					BACnetCalendarEntryType_DateRange:
						(* caclulate event entry size and write into data structure *)
						_pSpEventCalEntryRange^.nEntrySize :=	_cbTotalEntry
															+	SIZEOF(_pSpEventCalEntryRange^.stListEntry.eEventChoice)
															+	SIZEOF(_pSpEventCalEntryRange^.stListEntry.iEventPriority)
															+	SIZEOF(_pSpEventCalEntryRange^.stListEntry.nRes1)
															+	SIZEOF(_pSpEventCalEntryRange^.stListEntry.nRes2)
															+	SIZEOF(_pSpEventCalEntryRange^.stListEntry.stCalEntry);
						(* copy event data *)
						_pSpEventCalEntryRange^.stListEntry.eEventChoice := BACnetSpecialEventChoice_calendarEntry;
						_pSpEventCalEntryRange^.stListEntry.nRes1 := 0;
						_pSpEventCalEntryRange^.stListEntry.iEventPriority := stExceptSched.arrEntries[_iEntry].ePriority;
						_pSpEventCalEntryRange^.stListEntry.stCalEntry.eEntryChoice := BACnetCalendarEntryChoice_dateRange;
						_pSpEventCalEntryRange^.stListEntry.stCalEntry.nRes := 0;
						_pSpEventCalEntryRange^.stListEntry.stCalEntry.stStartDate := stExceptSched.arrEntries[_iEntry].stDate.stStart;
						_pSpEventCalEntryRange^.stListEntry.stCalEntry.stEndDate := stExceptSched.arrEntries[_iEntry].stDate.stEnd;

					BACnetCalendarEntryType_WeekNDay:
						(* caclulate event entry size and write into data structure *)
						_pSpEventCalEntryWnD^.nEntrySize :=	_cbTotalEntry
															+	SIZEOF(_pSpEventCalEntryWnD^.stListEntry.eEventChoice)
															+	SIZEOF(_pSpEventCalEntryWnD^.stListEntry.iEventPriority)
															+	SIZEOF(_pSpEventCalEntryWnD^.stListEntry.nRes1)
															+	SIZEOF(_pSpEventCalEntryWnD^.stListEntry.nRes2)
															+	SIZEOF(_pSpEventCalEntryWnD^.stListEntry.nRes3)
															+	SIZEOF(_pSpEventCalEntryWnD^.stListEntry.stCalEntry);
						(* copy event data *)
						_pSpEventCalEntryWnD^.stListEntry.eEventChoice := BACnetSpecialEventChoice_calendarEntry;
						_pSpEventCalEntryWnD^.stListEntry.nRes1 := 0;
						_pSpEventCalEntryWnD^.stListEntry.iEventPriority := stExceptSched.arrEntries[_iEntry].ePriority;
						_pSpEventCalEntryWnD^.stListEntry.stCalEntry.eEntryChoice := BACnetCalendarEntryChoice_weekNDay;
						_pSpEventCalEntryWnD^.stListEntry.stCalEntry.nRes1 := 0;
						_pSpEventCalEntryWnD^.stListEntry.stCalEntry.iDay := stExceptSched.arrEntries[_iEntry].stWeekNDay.iDay;
						_pSpEventCalEntryWnD^.stListEntry.stCalEntry.iMonth := stExceptSched.arrEntries[_iEntry].stWeekNDay.iMonth;
						_pSpEventCalEntryWnD^.stListEntry.stCalEntry.iWeekOfMonth := stExceptSched.arrEntries[_iEntry].stWeekNDay.iWeekOfMonth;

					BACnetCalendarEntryType_Ref:
						(* caclulate event entry size and write into data structure *)
						_pSpEventCalRef^.nEntrySize :=	_cbTotalEntry
													+	SIZEOF(_pSpEventCalRef^.stListEntry.eEventChoice)
													+	SIZEOF(_pSpEventCalRef^.stListEntry.iEventPriority)
													+	SIZEOF(_pSpEventCalRef^.stListEntry.nRes1)
													+	SIZEOF(_pSpEventCalRef^.stListEntry.nRes2)
													+	SIZEOF(_pSpEventCalRef^.stListEntry.nRes3)
													+	SIZEOF(_pSpEventCalRef^.stListEntry.nRes4)
													+	SIZEOF(_pSpEventCalRef^.stListEntry.tCalRef);
						(* copy event data *)
						_pSpEventCalRef^.stListEntry.eEventChoice := BACnetSpecialEventChoice_calendarReference;
						_pSpEventCalRef^.stListEntry.nRes1 := 0;
						_pSpEventCalRef^.stListEntry.iEventPriority := stExceptSched.arrEntries[_iEntry].ePriority;
						_pSpEventCalRef^.stListEntry.tCalRef := stExceptSched.arrEntries[_iEntry].stCalRef.tCalObjectId;

				END_CASE

				(* set next entry flag *)
				IF (_pOldEventEntrySize <> 0) THEN
					_pOldEventEntrySize^ := _pOldEventEntrySize^ + 16#80000000;
				END_IF

				(* next calendar entry *)
				_NextEvent();
			END_IF

		END_FOR

		(* send data *)
		_i := 19;

	19:
		IF _fbWriteProp.bExecute AND (NOT _fbWriteProp.bBusy) THEN
			(* check result *)
			_fbWriteProp.bExecute := FALSE;
			IF _fbWriteProp.bError THEN
				nErrorId := BACnet_ERR_ADS_Write;
			ELSE
				stExceptSched.nSet := stExceptSched.nSet +1;
			END_IF
			_i := 100;
		ELSE
			(* start ADS write *)
			_fbWriteProp.bExecute := TRUE;
		END_IF

	100: (* Done *)
		bDone := (nErrorId = BACnet_ERR_NO_ERROR);
		(* release ADS buffer *)
		stBACnet_AdsBuffer.iLocked := 0;
		(* release data array *)
		stExceptSched.bBusy := FALSE;
		(* go idle *)
		_i := 0;

END_CASE

(* set error flag *)
bError 	:= nErrorId > BACnet_ERR_NO_ERROR;
bBusy 	:= _i > 0;
END_FUNCTION_BLOCK
ACTION _NextEvent:
_bNextEvent := ((_pSpEventCalEntryDate^.nEntrySize AND 16#80000000) = 16#80000000);
_cbTmpSize := _F_BACnet_AlignedSize(_pSpEventCalEntryDate^.nEntrySize AND 16#7FFFFFFF) + SIZEOF(_pSpEventCalEntryDate^.nEntrySize) + SIZEOF(_pSpEventCalEntryDate^.nRes);
_pOldEventEntrySize		:= ADR(_pSpEventCalEntryDate^.nEntrySize);
_pSpEventCalEntryDate	:= _pSpEventCalEntryDate + _cbTmpSize;
_pSpEventCalEntryRange	:= _pSpEventCalEntryRange + _cbTmpSize;
_pSpEventCalEntryWnD	:= _pSpEventCalEntryWnD + _cbTmpSize;
_pSpEventCalRef			:= _pSpEventCalRef + _cbTmpSize;
_cbTotalBuf := _cbTotalBuf + _cbTmpSize;
_pOldTimeValue := 0;
END_ACTION
ACTION _NextTimeValue:
_bNextTimeValue := (_pTimeValue^.nEntrySize AND 16#80000000) = 16#80000000;
_cbTmpSize := 	(_F_BACnet_AlignedSize(_pTimeValue^.nEntrySize) AND 16#7FFFFFFF)
			+	SIZEOF(_pTimeValue^.nEntrySize)
			+	SIZEOF(_pTimeValue^.nRes);
_pOldTimeValue := _pTimeValue;
_pTimeValue := _pTimeValue + _cbTmpSize;
END_ACTION

(* POU FB_BACnet_ExceptionSchedulePropertyReal, ST *)
FUNCTION_BLOCK FB_BACnet_ExceptionSchedulePropertyReal
VAR_INPUT
	tObjectID			: T_BACnet_ObjectIdentifier := 16#FFFFFFFF;
	bAutoGet			: BOOL:=TRUE; (* TRUE = get data from property when ADS connection OR object ID changed *)
	bGet				: BOOL; (* FALSE --> TRUE = get data from property *)
	bSet				: BOOL; (* FALSE --> TRUE = set data into property *)
END_VAR
VAR_IN_OUT
	stExceptSched		: ST_BACnet_ExceptionScheduleReal;
	stAdsConn			: ST_BACnet_AdsConnection;
END_VAR
VAR_OUTPUT
	bDone				: BOOL;
	bBusy				: BOOL;
	bError				: BOOL;
	nErrorId			: UINT;
END_VAR
VAR
	_fbReadProp		: FB_BACnet_ReadProp;
	_fbWriteProp	: FB_BACnet_WriteProp;
	_i				: INT;
	_rtrigGet		: R_TRIG;
	_rtrigSet		: R_TRIG;

	_pOldEventEntrySize		: POINTER TO DWORD;
	_pSpEventCalEntryDate	: POINTER TO ST_BACnet_SpecialEventListCalEntryDate;
	_pSpEventCalEntryRange	: POINTER TO ST_BACnet_SpecialEventListCalEntryRange;
	_pSpEventCalEntryWnD	: POINTER TO ST_BACnet_SpecialEventListCalEntryWnD;
	_pSpEventCalRef			: POINTER TO ST_BACnet_SpecialEventListCalReference;
	_pTimeValue		: POINTER TO ST_BACnet_TimeValueList;
	_pOldTimeValue	: POINTER TO ST_BACnet_TimeValueList;

	_iEntry			: INT;
	_iTv			: INT;

	_bNextEvent		: BOOL;
	_bNextTimeValue	: BOOL;

	_cbTmpSize		: UDINT;
	_cbTotalEntry	: UDINT;
	_cbTotalBuf		: UDINT;
	_nAdsReloadOld	: USINT;
	_tObjectIDOld	: T_BACnet_ObjectIdentifier := 16#FFFFFFFF;

	_pReal			: POINTER TO REAL;
END_VAR
(*

Listheader:

typedef struct _ListEntryHdr
{
      DWORD nEntrySize;
      DWORD hdrInfo;
}ListEntryHdr, *PListEntryHdr;

#define ListAlignedSize(n)         (4*(((n)+3)/4))
#define FirstListEntry(p) ( (p)->nEntrySize == 0 )                          ? NULL:p
#define NextListEntry(p) ( ( ((p)->nEntrySize&0x80000000) == 0 ) ? NULL:(PBYTE)(p) + ( ListAlignedSize((p)->nEntrySize&~(0x80000000)) + sizeof(ListEntryHdr)) ) // +4 da für nEntrySize 4 Byte reserviert sind, HighBit ausmaskieren
#define ElemSize(p) ((p)->nEntrySize&(~0x80000000))
#define AlignedEntrySize(p) (ListAlignedSize((p)->nEntrySize&(~0x80000000)))

###################################################################

PropExceptionSchedule:

enum BACnetSpecialEventChoice
{
      calendarEntry,
      calendarReference,
      MaxBACnetSpecialEventChoice
};

typedef struct _BACnetCalendarEntry
{
      BACnetCalendarEntryChoice choice;
      union
      {
            BACnetDate              date;
            BACnetDateRange   dateRange;
            BACnetWeekNDay          weekNDay;
      };
}BACnetCalendarEntry, *PBACnetCalendarEntry;

enum BACnetValueChoice
{
      NullValue                    = 0,
      BoolValue                    = 1,
      UnsignedValue                = 2,
      SignedValue                  = 3,
      RealValue                    = 4,
      DoubleValue                  = 5,
      OctedStringValue        = 6,
      CharStringValue         = 7,
      ObjectIdentifierValue = 8,   // but DataType is 0x0C
      EnumerationValue        = 9,
      MaxBACnetValueChoice    = 10
};

typedef struct _BACnetValue  
{
      BACnetValueChoice choice;
      DWORD                        length;     // Alignment + Datenlänge die folgt
      union
      {
            BOOL                                     boolValue;
            FLOAT                                    realValue;
            DOUBLE                                   doubleValue;
            INT                                      signedValue;
            UINT                                     unsignedValue;
            BYTE*                                    pOctedStringValue; 
            CHAR*                                    pCharStringValue;
            BACnetObjectIdentifier  objectIdentifierValue;
            EnumerationValueType         enumerationValue;
      };
}BACnetValue, *PBACnetValue;

typedef struct _BACnetTimeValue
{
      BACnetTime time;
      DWORD  reserved;  // 64bit Alignment
      BACnetValue value;
}BACnetTimeValue, *PBACnetTimeValue;

typedef struct _BACnetTimeValueList
{
      DWORD nEntrySize; // 0x80000000 -> next entry
      DWORD reserved;
      BACnetTimeValue listEntry;
}BACnetTimeValueList, *PBACnetTimeValueList;

typedef struct _BACnetSpecialEvent
{
      BACnetSpecialEventChoice choice;
      union
      {
            BACnetCalendarEntry calendarEntry;
            BACnetObjectIdentifier calendarReference;
      };
      DWORD eventPriority; // DWORD due to alignment
      DWORD reserved;
      BACnetTimeValueList listOfTimeValues;
}BACnetSpecialEvent, *PBACnetSpecialEvent;

typedef struct _BACnetSpecialEventList
{
      DWORD nEntrySize; // 0x80000000 -> next entry
      DWORD reserved;
      BACnetSpecialEvent listEntry;
}BACnetSpecialEventList, *PBACnetSpecialEventList;

###################################################################

PropWeeklySchedule:

typedef struct _BACnetDailySchedule
{
      DWORD nEntrySize; // 0x80000000 -> next entry
      DWORD reserved;
      BACnetTimeValueList listEntry;
} BACnetDailySchedule, *PBACnetDailySchedule;

###################################################################

PropScheduleDefault / PropPresentValue

typedef struct _BACnetValueList
{
      DWORD nEntrySize; // 0x80000000 -> next entry
      DWORD reserved;
      BACnetValue listEntry;
} BACnetValueList, *PBACnetValueList;

###################################################################

*)

(* ADS read *)
_fbReadProp(
	BACnetDevicePort	:= stAdsConn.nAmsPort,
	bExecute			:= ,
	sNetId				:= stAdsConn.sAmsNetId,
	ObjectType			:= F_BACnet_GetObjType(tObjectID),
	PropertyID			:= BACnetPropertyIdentifier_ExceptionSchedule,
	DataType			:= BACnetDataType_SpecialEventList,
	ObjectInstance		:= F_BACnet_GetObjInstance(tObjectID),
	ptrValue			:= ADR(stBACnet_AdsBuffer.arrData),
	nLenValue			:= SIZEOF(stBACnet_AdsBuffer.arrData),
	bDone				=> ,
	bBusy				=> ,
	bError				=> ,
	nErrID				=> ,
	nProcessedLen		=> );

(* ADS write *)
_fbWriteProp(
	BACnetDevicePort	:= stAdsConn.nAmsPort,
	bExecute			:= ,
	sNetId				:= stAdsConn.sAmsNetId,
	ObjectType			:= F_BACnet_GetObjType(tObjectID),
	PropertyID			:= BACnetPropertyIdentifier_ExceptionSchedule,
	Priority			:= BACnetPriority_None,
	DataType			:= BACnetDataType_SpecialEventList,
	ObjectInstance		:= F_BACnet_GetObjInstance(tObjectID),
	ptrValue			:= ADR(stBACnet_AdsBuffer.arrData),
	nLenValue			:= _cbTotalBuf,
	bDone				=> ,
	bBusy				=> ,
	bError				=> ,
	nErrID				=> );

(* trigger start event *)
_rtrigGet(CLK:= bGet, Q=> );
_rtrigSet(CLK:= bSet, Q=> );

(* state machine *)
CASE _i OF

	0: (* Idle *)
		IF 		_rtrigGet.Q
			OR	_rtrigSet.Q
			OR	(		(		(_nAdsReloadOld <> stAdsConn.nReload)
							OR	(_tObjectIDOld <> tObjectID)
						)
					AND	bAutoGet
				)
			OR	stExceptSched.bReqGet
			OR	stExceptSched.bReqSet
		THEN
			IF (NOT stAdsConn.bValid) THEN
				(* ADS connection not valid *)
				nErrorId := BACnet_ERR_INVALID_ADS_CONN;
			ELSIF (NOT stAdsConn.bServer AND NOT stAdsConn.bClient) THEN
				(* not a server nor a client *)
				nErrorId := BACnet_ERR_ADS_NoServerClient;
			ELSE
				(* decide get or set *)
				IF _rtrigGet.Q OR stExceptSched.bReqGet  THEN
					_i := 1;
					stExceptSched.bReqGet := FALSE;
				ELSIF _rtrigSet.Q OR stExceptSched.bReqSet THEN
					_i := 11;
					stExceptSched.bReqSet := FALSE;
				ELSIF bAutoGet THEN
					_i := 1;
					stExceptSched.bReqGet := FALSE;
				END_IF
				nErrorId := BACnet_ERR_NO_ERROR;
				(* reset index *)
				_iEntry		:= 0;
				(* remind parameter *)
				_tObjectIDOld := tObjectID;
				_nAdsReloadOld := stAdsConn.nReload;
				(* lock data array *)
				stExceptSched.bBusy := TRUE;
			END_IF
			(* reset done flag *)
			bDone := FALSE;
		END_IF
		IF (NOT bGet) AND (NOT bSet) AND (NOT bAutoGet) THEN
			nErrorId := BACnet_ERR_NO_ERROR;
			bDone := FALSE;
		END_IF

	(* READ *)
	1: (* read object property data via ADS *)
		IF TestAndSet(stBACnet_AdsBuffer.bTestSet) THEN
			IF _fbReadProp.bExecute THEN
				IF _fbReadProp.bError THEN
					_i := 100;
					nErrorId := BACnet_ERR_ADS_Read;
					_fbReadProp.bExecute := FALSE;
				ELSIF (NOT _fbReadProp.bBusy) THEN
					_i := 2;
					_fbReadProp.bExecute := FALSE;
					(* prepare pointer *)
					_pSpEventCalEntryDate	:= ADR(stBACnet_AdsBuffer.arrData);
					_pSpEventCalEntryRange	:= ADR(stBACnet_AdsBuffer.arrData);
					_pSpEventCalEntryWnD	:= ADR(stBACnet_AdsBuffer.arrData);
					_pSpEventCalRef			:= ADR(stBACnet_AdsBuffer.arrData);
					(* clear output data *)
					MEMSET(ADR(stExceptSched.arrEntries), 0, SIZEOF(stExceptSched.arrEntries));
					_cbTotalBuf := 0;
					_bNextEvent := TRUE;
				END_IF

			ELSIF (stBACnet_AdsBuffer.iLocked = 0) THEN
				_fbReadProp.bExecute := TRUE;
				(* lock global ADS buffer *)
				stBACnet_AdsBuffer.iLocked := SIZEOF(stBACnet_AdsBuffer.arrData);
			END_IF

			(* release temporary task lock *)
			stBACnet_AdsBuffer.bTestSet := FALSE;
		END_IF

	2: (* select event entry *)
		(* more events? *)
		IF (NOT _bNextEvent) THEN
			(* no more events, exit *)
			_i := 4;
		ELSE
			_i := 3;
			(* check if local buffer is full *)
			IF _iEntry > BACnet_MaxExSchEntries THEN
				_i := 4; (* maximum entries reached --> finished *)
			ELSIF ((_pSpEventCalEntryDate^.nEntrySize AND 16#7FFFFFFF) > 0) THEN
				(* initialize first entry *)
				stExceptSched.arrEntries[_iEntry].eEntryType := BACnetCalendarEntryType_None;

				CASE _pSpEventCalEntryDate^.stListEntry.eEventChoice OF

					BACnetSpecialEventChoice_calendarReference:
						_pTimeValue := ADR(_pSpEventCalRef^.stListEntry.stListOfTimeValues);
						stExceptSched.arrEntries[_iEntry].eEntryType := BACnetCalendarEntryType_Ref;
						stExceptSched.arrEntries[_iEntry].stCalRef.tCalObjectId := _pSpEventCalRef^.stListEntry.tCalRef;
						stExceptSched.arrEntries[_iEntry].ePriority := DWORD_TO_INT(_pSpEventCalRef^.stListEntry.iEventPriority);

					BACnetSpecialEventChoice_calendarEntry:
						CASE _pSpEventCalEntryDate^.stListEntry.stCalEntry.eEntryChoice OF
							BACnetCalendarEntryChoice_date:
								_pTimeValue := ADR(_pSpEventCalEntryDate^.stListEntry.stListOfTimeValues);
								stExceptSched.arrEntries[_iEntry].eEntryType := BACnetCalendarEntryType_Date;
								stExceptSched.arrEntries[_iEntry].stDate.stStart := _pSpEventCalEntryDate^.stListEntry.stCalEntry.stDate;
								stExceptSched.arrEntries[_iEntry].stDate.stEnd := _pSpEventCalEntryDate^.stListEntry.stCalEntry.stDate;
								stExceptSched.arrEntries[_iEntry].ePriority := DWORD_TO_INT(_pSpEventCalEntryDate^.stListEntry.iEventPriority);

							BACnetCalendarEntryChoice_dateRange:
								_pTimeValue := ADR(_pSpEventCalEntryRange^.stListEntry.stListOfTimeValues);
								stExceptSched.arrEntries[_iEntry].eEntryType := BACnetCalendarEntryType_DateRange;
								stExceptSched.arrEntries[_iEntry].stDate.stStart := _pSpEventCalEntryRange^.stListEntry.stCalEntry.stStartDate;
								stExceptSched.arrEntries[_iEntry].stDate.stEnd := _pSpEventCalEntryRange^.stListEntry.stCalEntry.stEndDate;
								stExceptSched.arrEntries[_iEntry].ePriority := DWORD_TO_INT(_pSpEventCalEntryRange^.stListEntry.iEventPriority);

							BACnetCalendarEntryChoice_weekNDay:
								_pTimeValue := ADR(_pSpEventCalEntryWnD^.stListEntry.stListOfTimeValues);
								stExceptSched.arrEntries[_iEntry].eEntryType := BACnetCalendarEntryType_WeekNDay;
								stExceptSched.arrEntries[_iEntry].stWeekNDay.iMonth := _pSpEventCalEntryWnD^.stListEntry.stCalEntry.iMonth;
								stExceptSched.arrEntries[_iEntry].stWeekNDay.iWeekOfMonth := _pSpEventCalEntryWnD^.stListEntry.stCalEntry.iWeekOfMonth;
								stExceptSched.arrEntries[_iEntry].stWeekNDay.iDay := _pSpEventCalEntryWnD^.stListEntry.stCalEntry.iDay;
								stExceptSched.arrEntries[_iEntry].ePriority := DWORD_TO_INT(_pSpEventCalEntryWnD^.stListEntry.iEventPriority);

							ELSE
								(* unknown entry choice *)
								nErrorId := BACnet_ERR_UnknownEntryChoice;
								_i := 100;
						END_CASE
					ELSE
						(* unknown event choice *)
						nErrorId := BACnet_ERR_UnknownEventChoice;
						_i := 100;
				END_CASE
			ELSE
				(* mark as invalid *)
				stExceptSched.arrEntries[_iEntry].eEntryType := BACnetCalendarEntryType_None;
			END_IF
		END_IF
		(* reset time value index *)
		_iTv := 0;

	3: (* scan time value list *)
		(* preset next time value flag *)
		_bNextTimeValue := TRUE;
		(* loop till all time values are parsed *)
		WHILE _bNextTimeValue AND _pTimeValue <> 0 DO
			IF ((_pTimeValue^.nEntrySize AND 16#7FFFFFFF) > 0) AND (_iTv <= BACnet_MaxTimeValues) THEN
				(* time value data available - is it a real type? *)
				IF		_pTimeValue^.stListEntry.stValue.eValueChoice = BACnetDataType_Real
					OR	_pTimeValue^.stListEntry.stValue.eValueChoice = BACnetDataType_Null
				THEN
					(* decide entry type *)
					CASE stExceptSched.arrEntries[_iEntry].eEntryType OF
						BACnetCalendarEntryType_Date,
						BACnetCalendarEntryType_DateRange:
							stExceptSched.arrEntries[_iEntry].arrTimeValue[_iTv].bValid := TRUE;
							stExceptSched.arrEntries[_iEntry].arrTimeValue[_iTv].stTime := _pTimeValue^.stListEntry.stTime;
							stExceptSched.arrEntries[_iEntry].arrTimeValue[_iTv].eType := _pTimeValue^.stListEntry.stValue.eValueChoice;
							IF _pTimeValue^.stListEntry.stValue.cbData = 4 THEN
								MEMCPY(	ADR(stExceptSched.arrEntries[_iEntry].arrTimeValue[_iTv].rValue),
										ADR(_pTimeValue^.stListEntry.stValue.nData),
										SIZEOF(stExceptSched.arrEntries[_iEntry].arrTimeValue[_iTv].rValue)
								);
							ELSE
								stExceptSched.arrEntries[_iEntry].arrTimeValue[_iTv].rValue := F_BACnet_NAN();
							END_IF
							_iTv := _iTv +1;

						BACnetCalendarEntryType_WeekNDay:
							stExceptSched.arrEntries[_iEntry].arrTimeValue[_iTv].bValid := TRUE;
							stExceptSched.arrEntries[_iEntry].arrTimeValue[_iTv].stTime := _pTimeValue^.stListEntry.stTime;
							stExceptSched.arrEntries[_iEntry].arrTimeValue[_iTv].eType := _pTimeValue^.stListEntry.stValue.eValueChoice;
							IF _pTimeValue^.stListEntry.stValue.cbData = 4 THEN
								MEMCPY(	ADR(stExceptSched.arrEntries[_iEntry].arrTimeValue[_iTv].rValue),
										ADR(_pTimeValue^.stListEntry.stValue.nData),
										SIZEOF(stExceptSched.arrEntries[_iEntry].arrTimeValue[_iTv].rValue)
								);
							ELSE
								stExceptSched.arrEntries[_iEntry].arrTimeValue[_iTv].rValue := F_BACnet_NAN();
							END_IF
							_iTv := _iTv +1;

						BACnetCalendarEntryType_Ref:
							stExceptSched.arrEntries[_iEntry].arrTimeValue[_iTv].bValid := TRUE;
							stExceptSched.arrEntries[_iEntry].arrTimeValue[_iTv].stTime := _pTimeValue^.stListEntry.stTime;
							stExceptSched.arrEntries[_iEntry].arrTimeValue[_iTv].eType := _pTimeValue^.stListEntry.stValue.eValueChoice;
							IF _pTimeValue^.stListEntry.stValue.cbData = 4 THEN
								MEMCPY(	ADR(stExceptSched.arrEntries[_iEntry].arrTimeValue[_iTv].rValue),
										ADR(_pTimeValue^.stListEntry.stValue.nData),
										SIZEOF(stExceptSched.arrEntries[_iEntry].arrTimeValue[_iTv].rValue)
								);
							ELSE
								stExceptSched.arrEntries[_iEntry].arrTimeValue[_iTv].rValue := F_BACnet_NAN();
							END_IF
							_iTv := _iTv +1;

					END_CASE

				ELSE
					(* unsupported data type *);
				END_IF

			END_IF

			(* empty entry size or data buffer full, next time value entry *)
			_NextTimeValue();

		END_WHILE

		(* count *)(*
		IF _iTv > 0 THEN
			_iEntry := _iEntry +1;
		END_IF*)
		_iEntry := _iEntry +1;

		(* next event entry *)
		_NextEvent();
		_i := 2;

	4: (* data read and parsed successful *)
		stExceptSched.nGet := stExceptSched.nGet +1;
		_i := 100;

	11: (* lock global ADS buffer *)
		IF TestAndSet(stBACnet_AdsBuffer.bTestSet) THEN
			IF stBACnet_AdsBuffer.iLocked = 0 THEN
				stBACnet_AdsBuffer.iLocked := SIZEOF(stBACnet_AdsBuffer.arrData);
				(* initalize total size counter *)
				_cbTotalBuf := 0;
				(* prepare pointer *)
				_pSpEventCalEntryDate	:= ADR(stBACnet_AdsBuffer.arrData);
				_pSpEventCalEntryRange	:= ADR(stBACnet_AdsBuffer.arrData);
				_pSpEventCalEntryWnD	:= ADR(stBACnet_AdsBuffer.arrData);
				_pSpEventCalRef			:= ADR(stBACnet_AdsBuffer.arrData);
				_pOldEventEntrySize		:= 0;
				(* loop against input data *)
				_i := 12;
			END_IF
			(* release temporary task lock *)
			stBACnet_AdsBuffer.bTestSet := FALSE;
		END_IF

	12: (* write calendar entries date/date range *)
		FOR _iEntry := 0 TO BACnet_MaxExSchEntries DO

			_pOldTimeValue	:= 0;
			_cbTotalEntry	:= 0;

			IF stExceptSched.arrEntries[_iEntry].eEntryType <> BACnetCalendarEntryType_None THEN
				(* valid entry *)
				CASE stExceptSched.arrEntries[_iEntry].eEntryType OF

					BACnetCalendarEntryType_Date,
					BACnetCalendarEntryType_DateRange:
						(* set special entry choice *)
						IF stExceptSched.arrEntries[_iEntry].eEntryType = BACnetCalendarEntryType_Date THEN
							_pSpEventCalEntryDate^.stListEntry.eEventChoice := BACnetSpecialEventChoice_calendarEntry;
							_pSpEventCalEntryDate^.stListEntry.nRes1 := 0;
							(* set time value pointer *)
							_pTimeValue := ADR(_pSpEventCalEntryDate^.stListEntry.stListOfTimeValues);
						ELSE
							_pSpEventCalEntryRange^.stListEntry.eEventChoice := BACnetSpecialEventChoice_calendarEntry;
							_pSpEventCalEntryRange^.stListEntry.nRes1 := 0;
							(* set time value pointer *)
							_pTimeValue := ADR(_pSpEventCalEntryRange^.stListEntry.stListOfTimeValues);
						END_IF

					BACnetCalendarEntryType_WeekNDay:
						(* set special entry choice *)
						_pSpEventCalEntryWnD^.stListEntry.eEventChoice := BACnetSpecialEventChoice_calendarEntry;
						_pSpEventCalEntryWnD^.stListEntry.nRes1 := 0;
						(* set time value pointer *)
						_pTimeValue := ADR(_pSpEventCalEntryWnD^.stListEntry.stListOfTimeValues);

					BACnetCalendarEntryType_Ref:
						(* set special entry choice *)
						_pSpEventCalRef^.stListEntry.eEventChoice := BACnetSpecialEventChoice_calendarReference;
						_pSpEventCalRef^.stListEntry.nRes1 := 0;
						(* set time value pointer *)
						_pTimeValue := ADR(_pSpEventCalRef^.stListEntry.stListOfTimeValues);

				END_CASE


				(* loop against time values *)
				FOR _iTv := 0 TO BACnet_MaxTimeValues DO

					(* valid entry? *)
					IF stExceptSched.arrEntries[_iEntry].arrTimeValue[_iTv].bValid THEN
						(* copy time *)
						_pTimeValue^.stListEntry.stTime := stExceptSched.arrEntries[_iEntry].arrTimeValue[_iTv].stTime;
						_pReal := ADR(_pTimeValue^.stListEntry.stValue.nData);
						_pReal^ := 0.0; (* clear data *)
						(* decide between None and Real type *)
						IF stExceptSched.arrEntries[_iEntry].arrTimeValue[_iTv].eType = BACnetDataType_Real THEN
							(* REAL type *)
							_pTimeValue^.stListEntry.stValue.eValueChoice := BACnetDataType_Real;
							_pTimeValue^.stListEntry.stValue.nRes1 := 0;
							_pTimeValue^.stListEntry.stValue.cbData := SIZEOF(stExceptSched.arrEntries[_iEntry].arrTimeValue[_iTv].rValue);
							MEMCPY(	_pReal,
									ADR(stExceptSched.arrEntries[_iEntry].arrTimeValue[_iTv].rValue),
									MIN(SIZEOF(_pReal^), _pTimeValue^.stListEntry.stValue.cbData)
							);
						ELSE
							(* other or NONE type *)
							_pTimeValue^.stListEntry.stValue.eValueChoice := BACnetDataType_Null;
							_pTimeValue^.stListEntry.stValue.nRes1 := 0;
							_pTimeValue^.stListEntry.stValue.cbData := 0;
						END_IF

						(* calculate time-value entry size *)
						_pTimeValue^.nEntrySize :=	_pTimeValue^.stListEntry.stValue.cbData
												+	SIZEOF(_pTimeValue^.stListEntry.nRes)
												+	SIZEOF(_pTimeValue^.stListEntry.stTime)
												+	SIZEOF(_pTimeValue^.stListEntry.stValue.cbData)
												+	SIZEOF(_pTimeValue^.stListEntry.stValue.eValueChoice)
												+	SIZEOF(_pTimeValue^.stListEntry.stValue.nRes1);

						IF (_iTv > 0 AND _pOldTimeValue <> 0) THEN
							(* next entry flag *)
							_pOldTimeValue^.nEntrySize := _pOldTimeValue^.nEntrySize + 16#80000000;
						END_IF

						(* update time value pointer *)
						_NextTimeValue();

						(* ...and add to total entry size counter *)
						_cbTotalEntry := _cbTotalEntry + _cbTmpSize;

					ELSE
						(* clear entry *)
						_pTimeValue^.nEntrySize := 0;
						_pTimeValue^.stListEntry.stValue.cbData := 0;
					END_IF

				END_FOR

				(* check if time value list is empty *)
				IF _cbTotalEntry = 0 THEN
					(* no time values, set default size *)
					_cbTotalEntry := SIZEOF(_pTimeValue^.nEntrySize) + SIZEOF(_pTimeValue^.nRes);
				END_IF

				(* caclulate event entry size *)
				CASE stExceptSched.arrEntries[_iEntry].eEntryType OF

					BACnetCalendarEntryType_Date:
						(* caclulate event entry size and write into data structure *)
						_pSpEventCalEntryDate^.nEntrySize :=	_cbTotalEntry
															+	SIZEOF(_pSpEventCalEntryDate^.stListEntry.eEventChoice)
															+	SIZEOF(_pSpEventCalEntryDate^.stListEntry.iEventPriority)
															+	SIZEOF(_pSpEventCalEntryDate^.stListEntry.nRes1)
															+	SIZEOF(_pSpEventCalEntryDate^.stListEntry.nRes2)
															+	SIZEOF(_pSpEventCalEntryDate^.stListEntry.nRes3)
															+	SIZEOF(_pSpEventCalEntryDate^.stListEntry.stCalEntry);
						(* copy event data *)
						_pSpEventCalEntryDate^.stListEntry.eEventChoice := BACnetSpecialEventChoice_calendarEntry;
						_pSpEventCalEntryDate^.stListEntry.nRes1 := 0;
						_pSpEventCalEntryDate^.stListEntry.iEventPriority := stExceptSched.arrEntries[_iEntry].ePriority;
						_pSpEventCalEntryDate^.stListEntry.stCalEntry.eEntryChoice := BACnetCalendarEntryChoice_date;
						_pSpEventCalEntryDate^.stListEntry.stCalEntry.nRes := 0;
						_pSpEventCalEntryDate^.stListEntry.stCalEntry.stDate := stExceptSched.arrEntries[_iEntry].stDate.stStart;

					BACnetCalendarEntryType_DateRange:
						(* caclulate event entry size and write into data structure *)
						_pSpEventCalEntryRange^.nEntrySize :=	_cbTotalEntry
															+	SIZEOF(_pSpEventCalEntryRange^.stListEntry.eEventChoice)
															+	SIZEOF(_pSpEventCalEntryRange^.stListEntry.iEventPriority)
															+	SIZEOF(_pSpEventCalEntryRange^.stListEntry.nRes1)
															+	SIZEOF(_pSpEventCalEntryRange^.stListEntry.nRes2)
															+	SIZEOF(_pSpEventCalEntryRange^.stListEntry.stCalEntry);
						(* copy event data *)
						_pSpEventCalEntryRange^.stListEntry.eEventChoice := BACnetSpecialEventChoice_calendarEntry;
						_pSpEventCalEntryRange^.stListEntry.nRes1 := 0;
						_pSpEventCalEntryRange^.stListEntry.iEventPriority := stExceptSched.arrEntries[_iEntry].ePriority;
						_pSpEventCalEntryRange^.stListEntry.stCalEntry.eEntryChoice := BACnetCalendarEntryChoice_dateRange;
						_pSpEventCalEntryRange^.stListEntry.stCalEntry.nRes := 0;
						_pSpEventCalEntryRange^.stListEntry.stCalEntry.stStartDate := stExceptSched.arrEntries[_iEntry].stDate.stStart;
						_pSpEventCalEntryRange^.stListEntry.stCalEntry.stEndDate := stExceptSched.arrEntries[_iEntry].stDate.stEnd;

					BACnetCalendarEntryType_WeekNDay:
						(* caclulate event entry size and write into data structure *)
						_pSpEventCalEntryWnD^.nEntrySize :=	_cbTotalEntry
															+	SIZEOF(_pSpEventCalEntryWnD^.stListEntry.eEventChoice)
															+	SIZEOF(_pSpEventCalEntryWnD^.stListEntry.iEventPriority)
															+	SIZEOF(_pSpEventCalEntryWnD^.stListEntry.nRes1)
															+	SIZEOF(_pSpEventCalEntryWnD^.stListEntry.nRes2)
															+	SIZEOF(_pSpEventCalEntryWnD^.stListEntry.nRes3)
															+	SIZEOF(_pSpEventCalEntryWnD^.stListEntry.stCalEntry);
						(* copy event data *)
						_pSpEventCalEntryWnD^.stListEntry.eEventChoice := BACnetSpecialEventChoice_calendarEntry;
						_pSpEventCalEntryWnD^.stListEntry.nRes1 := 0;
						_pSpEventCalEntryWnD^.stListEntry.iEventPriority := stExceptSched.arrEntries[_iEntry].ePriority;
						_pSpEventCalEntryWnD^.stListEntry.stCalEntry.eEntryChoice := BACnetCalendarEntryChoice_weekNDay;
						_pSpEventCalEntryWnD^.stListEntry.stCalEntry.nRes1 := 0;
						_pSpEventCalEntryWnD^.stListEntry.stCalEntry.iDay := stExceptSched.arrEntries[_iEntry].stWeekNDay.iDay;
						_pSpEventCalEntryWnD^.stListEntry.stCalEntry.iMonth := stExceptSched.arrEntries[_iEntry].stWeekNDay.iMonth;
						_pSpEventCalEntryWnD^.stListEntry.stCalEntry.iWeekOfMonth := stExceptSched.arrEntries[_iEntry].stWeekNDay.iWeekOfMonth;

					BACnetCalendarEntryType_Ref:
						(* caclulate event entry size and write into data structure *)
						_pSpEventCalRef^.nEntrySize :=	_cbTotalEntry
													+	SIZEOF(_pSpEventCalRef^.stListEntry.eEventChoice)
													+	SIZEOF(_pSpEventCalRef^.stListEntry.iEventPriority)
													+	SIZEOF(_pSpEventCalRef^.stListEntry.nRes1)
													+	SIZEOF(_pSpEventCalRef^.stListEntry.nRes2)
													+	SIZEOF(_pSpEventCalRef^.stListEntry.nRes3)
													+	SIZEOF(_pSpEventCalRef^.stListEntry.nRes4)
													+	SIZEOF(_pSpEventCalRef^.stListEntry.tCalRef);
						(* copy event data *)
						_pSpEventCalRef^.stListEntry.eEventChoice := BACnetSpecialEventChoice_calendarReference;
						_pSpEventCalRef^.stListEntry.nRes1 := 0;
						_pSpEventCalRef^.stListEntry.iEventPriority := stExceptSched.arrEntries[_iEntry].ePriority;
						_pSpEventCalRef^.stListEntry.tCalRef := stExceptSched.arrEntries[_iEntry].stCalRef.tCalObjectId;

				END_CASE

				(* set next entry flag *)
				IF (_pOldEventEntrySize <> 0) THEN
					_pOldEventEntrySize^ := _pOldEventEntrySize^ + 16#80000000;
				END_IF

				(* next calendar entry *)
				_NextEvent();
			END_IF

		END_FOR

		(* send data *)
		_i := 19;

	19:
		IF _fbWriteProp.bExecute AND (NOT _fbWriteProp.bBusy) THEN
			(* check result *)
			_fbWriteProp.bExecute := FALSE;
			IF _fbWriteProp.bError THEN
				nErrorId := BACnet_ERR_ADS_Write;
			ELSE
				stExceptSched.nSet := stExceptSched.nSet +1;
			END_IF
			_i := 100;
		ELSE
			(* start ADS write *)
			_fbWriteProp.bExecute := TRUE;
		END_IF

	100: (* Done *)
		bDone := (nErrorId = BACnet_ERR_NO_ERROR);
		(* release ADS buffer *)
		stBACnet_AdsBuffer.iLocked := 0;
		(* release data array *)
		stExceptSched.bBusy := FALSE;
		(* go idle *)
		_i := 0;

END_CASE

(* set error flag *)
bError 	:= nErrorId > BACnet_ERR_NO_ERROR;
bBusy 	:= _i > 0;
END_FUNCTION_BLOCK
ACTION _NextEvent:
_bNextEvent := ((_pSpEventCalEntryDate^.nEntrySize AND 16#80000000) = 16#80000000);
_cbTmpSize := _F_BACnet_AlignedSize(_pSpEventCalEntryDate^.nEntrySize AND 16#7FFFFFFF) + SIZEOF(_pSpEventCalEntryDate^.nEntrySize) + SIZEOF(_pSpEventCalEntryDate^.nRes);
_pOldEventEntrySize		:= ADR(_pSpEventCalEntryDate^.nEntrySize);
_pSpEventCalEntryDate	:= _pSpEventCalEntryDate + _cbTmpSize;
_pSpEventCalEntryRange	:= _pSpEventCalEntryRange + _cbTmpSize;
_pSpEventCalEntryWnD	:= _pSpEventCalEntryWnD + _cbTmpSize;
_pSpEventCalRef			:= _pSpEventCalRef + _cbTmpSize;
_cbTotalBuf := _cbTotalBuf + _cbTmpSize;
_pOldTimeValue := 0;
END_ACTION
ACTION _NextTimeValue:
_bNextTimeValue := (_pTimeValue^.nEntrySize AND 16#80000000) = 16#80000000;
_cbTmpSize := 	(_F_BACnet_AlignedSize(_pTimeValue^.nEntrySize) AND 16#7FFFFFFF)
			+	SIZEOF(_pTimeValue^.nEntrySize)
			+	SIZEOF(_pTimeValue^.nRes);
_pOldTimeValue := _pTimeValue;
_pTimeValue := _pTimeValue + _cbTmpSize;
END_ACTION

(* POU FB_BACnet_File, ST *)
FUNCTION_BLOCK FB_BACnet_File
VAR_IN_OUT
	Device	: FB_BACnet_Device;
END_VAR
VAR_OUTPUT
	bReady			: BOOL;
	nFileSize		: UDINT;
	bError			: BOOL;
	nErrorId		: UINT;
END_VAR
VAR
	_FileSize 			AT%I*: UDINT; 	(* ~(BACnet_FileSize 				:		: )
					   						(BACnet_ObjectType 				: FILE	: )	*)
	_nUpdateCount		: UDINT := 0;
END_VAR
(* update server device *)
IF (Device._nUpdateCount = _nUpdateCount) THEN
	Device();
END_IF
(* remind current number of update counter *)
_nUpdateCount := Device._nUpdateCount;

IF Device.bOperational THEN
	(* ready state *)
	bReady := TRUE;
	nErrorId := BACnet_ERR_NO_ERROR;
	nFileSize := _FileSize;
ELSE
	(* server device not ready, reset local ready also *)
	bReady := FALSE;
	nErrorId := BACnet_ERR_OPERATIONAL;
END_IF
(* set error flag *)
bError := (nErrorId <> BACnet_ERR_NO_ERROR);
END_FUNCTION_BLOCK

(* POU FB_BACnet_File_EX, ST *)
FUNCTION_BLOCK FB_BACnet_File_EX
VAR_IN_OUT
	Device				: FB_BACnet_Device;
END_VAR
VAR_OUTPUT
	bReady				: BOOL;
	nFileSize			: UDINT;
	tObjectID			: T_BACnet_ObjectIdentifier := 16#FFFFFFFF;
	bError				: BOOL;
	nErrorId			: UINT;
END_VAR
VAR
	_FileSize 			AT%I*: UDINT; 	(* ~(BACnet_FileSize 		:		: )
					   						(BACnet_ObjectType 		: FILE	: )	*)
	_ObjectId AT%I*: DWORD;				(* ~(BACnet_ObjectIdentifier:		: LINK) *)
	_nUpdateCount		: UDINT := 0;
END_VAR
(* update server device *)
IF (Device._nUpdateCount = _nUpdateCount) THEN
	Device();
END_IF
(* remind current number of update counter *)
_nUpdateCount := Device._nUpdateCount;

IF (F_BACnet_GetObjType(_ObjectId) <> BACnetObjectType_File) THEN
	(* wrong mapping / invalid object ID *)
	IF _ObjectId = 0 THEN
		nErrorId := BACnet_ERR_WRONG_MAPPING;
	ELSE
		nErrorId := BACnet_ERR_INVALID_OBJECTID;
	END_IF
	bReady := FALSE;
	tObjectID := 16#FFFFFFFF;

ELSIF Device.bOperational THEN
	(* ready state *)
	bReady := TRUE;
	nErrorId := BACnet_ERR_NO_ERROR;
	nFileSize := _FileSize;
	tObjectID := _ObjectId;

ELSE
	(* server device not ready, reset local ready also *)
	bReady := FALSE;
	nErrorId := BACnet_ERR_OPERATIONAL;
END_IF
(* set error flag *)
bError := (nErrorId <> BACnet_ERR_NO_ERROR);
END_FUNCTION_BLOCK

(* POU FB_BACnet_GetDiagInfo, ST *)
FUNCTION_BLOCK FB_BACnet_GetDiagInfo
VAR_INPUT
	sNetId		: T_AmsNetId;
	bExecute	: BOOL;
	tTimeout	: TIME := BACnet_ADSTimeOut;
END_VAR
VAR_OUTPUT
	bBusy		: BOOL;
	bError		: BOOL;
	nErrID		: UDINT;
	stInfo		: ST_BACnet_Diagnosis;
END_VAR
VAR
	_fbAdsRead	: ADSREAD;
END_VAR
(* call ADS read function to receive info data *)
_fbAdsRead(
	NETID	:= sNetId,
	PORT	:= 16#FFFF, (* ADS port of BACnet device adapter *)
	IDXGRP	:= 16#8000000F,
	IDXOFFS	:= 16#0000,
	LEN		:= SIZEOF(stInfo),
	DESTADDR:= ADR(stInfo),
	READ	:= bExecute,
	TMOUT	:= tTimeout,
	BUSY	=> bBusy,
	ERR		=> bError,
	ERRID	=> nErrID);
END_FUNCTION_BLOCK

(* POU FB_BACnet_Group, ST *)
FUNCTION_BLOCK FB_BACnet_Group
VAR_IN_OUT
	Device	: FB_BACnet_Device;
END_VAR
VAR_OUTPUT
	bReady			: BOOL;
	bError			: BOOL;
	nErrorId		: UINT;
END_VAR
VAR
	_nUpdateCount : UDINT := 0; (* ~(BACNET_OBJECTTYPE : GROUP : NOLINK)	*)
END_VAR
(* update server device *)
IF (Device._nUpdateCount = _nUpdateCount) THEN
	Device();
END_IF
(* remind current number of update counter *)
_nUpdateCount := Device._nUpdateCount;

IF Device.bOperational THEN
	(* ready state *)
	bReady := TRUE;
	nErrorId := BACnet_ERR_NO_ERROR;
ELSE
	(* server device not ready, reset local ready also *)
	bReady := FALSE;
	nErrorId := BACnet_ERR_OPERATIONAL;
END_IF
(* set error flag *)
bError := (nErrorId <> BACnet_ERR_NO_ERROR);
END_FUNCTION_BLOCK

(* POU FB_BACnet_Group_EX, ST *)
FUNCTION_BLOCK FB_BACnet_Group_EX
VAR_IN_OUT
	Device				: FB_BACnet_Device;
END_VAR
VAR_OUTPUT
	bReady				: BOOL;
	tObjectID			: T_BACnet_ObjectIdentifier := 16#FFFFFFFF;
	bError				: BOOL;
	nErrorId			: UINT;
END_VAR
VAR
	_ObjectId AT%I*: DWORD;		(* ~(BACnet_ObjectIdentifier:		: LINK)
									(BACNET_OBJECTTYPE		: GROUP : ) *)
	_nUpdateCount : UDINT := 0;
END_VAR
(* update server device *)
IF (Device._nUpdateCount = _nUpdateCount) THEN
	Device();
END_IF
(* remind current number of update counter *)
_nUpdateCount := Device._nUpdateCount;

IF (F_BACnet_GetObjType(_ObjectId) <> BACnetObjectType_Group) THEN
	(* wrong mapping / invalid object ID *)
	IF _ObjectId = 0 THEN
		nErrorId := BACnet_ERR_WRONG_MAPPING;
	ELSE
		nErrorId := BACnet_ERR_INVALID_OBJECTID;
	END_IF
	bReady := FALSE;
	tObjectID := 16#FFFFFFFF;

ELSIF Device.bOperational THEN
	(* ready state *)
	bReady := TRUE;
	nErrorId := BACnet_ERR_NO_ERROR;
	tObjectID := _ObjectId;
ELSE
	(* server device not ready, reset local ready also *)
	bReady := FALSE;
	nErrorId := BACnet_ERR_OPERATIONAL;
END_IF
(* set error flag *)
bError := (nErrorId <> BACnet_ERR_NO_ERROR);
END_FUNCTION_BLOCK

(* POU FB_BACnet_LogBufferProperty, ST *)
FUNCTION_BLOCK FB_BACnet_LogBufferProperty
VAR_INPUT
	tObjectID			: T_BACnet_ObjectIdentifier := 16#FFFFFFFF;
	bAutoGet			: BOOL:=TRUE; (* TRUE = get data from property when ADS connection OR object ID changed *)
	bGet				: BOOL; (* FALSE --> TRUE = get data from property *)
	stStartTime			: ST_BACnet_DateTime := (
							stDate := (nYear := 16#FF, nMonth := 16#FF, nDay := 16#FF),
							stTime := (nHour := 16#FF, nMinute := 16#FF, nSecond := 16#FF, nHundredths := 16#FF)
							); (* Log record beginning from time stStartTime ... (16#FF = unspecified) *)
	stEndTime			: ST_BACnet_DateTime := (
							stDate := (nYear := 16#FF, nMonth := 16#FF, nDay := 16#FF),
							stTime := (nHour := 16#FF, nMinute := 16#FF, nSecond := 16#FF, nHundredths := 16#FF)
							); (* till end time stEndTime (16#FF = unspecified) *)
END_VAR
VAR_IN_OUT
	stAdsConn			: ST_BACnet_AdsConnection;
END_VAR
VAR_OUTPUT
	bDone				: BOOL;
	bBusy				: BOOL;
	bError				: BOOL;
	nErrorId			: UINT;
	stLogBuffer			: ST_BACnet_LogBufferReal;
END_VAR
VAR CONSTANT
	_stMaxTime			: ST_BACnet_Time := (nHour := 23, nMinute := 59, nSecond := 59, nHundredths := 99);
	_stMaxDate			: st_bacnet_date := (nYear := 254, nMonth := 12, nDay := 31, nDayOfWeek := 7);
END_VAR
VAR
	_fbReadProp		: FB_BACnet_ReadProp;
	_fbObjDesc		: FB_BACnet_DescriptionProperty;
	_fbObjName		: FB_BACnet_ObjectNameProperty;
	_i				: INT;
	_rtrigGet		: R_TRIG;

	_pAdsBuf		: POINTER TO BYTE;
	_pLbRecordList	: POINTER TO ST_BACnet_LogRecordList; (* Log buffer - record list *)
	_pLrDatumList	: POINTER TO ST_BACnet_LogDatumList; (* Log record entry - datum list *)

	_iEntry			: INT;

	_bNextRecord	: BOOL;
	_bNextDatum		: BOOL;

	_cbTmpSize		: UDINT;
	_cbTotalBuf		: UDINT;
	_nAdsReloadOld	: USINT;
	_tObjectIDOld	: T_BACnet_ObjectIdentifier := 16#FFFFFFFF;

	_arrRecords		: ARRAY[0..BACnet_MaxLogBufferEntries] OF POINTER TO ST_BACnet_LogRecordList;
	_iNextRecPos	: UDINT;
	_nRecCount		: UDINT;
	_iRec			: UDINT;
	_nMaxSeq		: DWORD; (* max. found sequence no. *)

	_pReal			: POINTER TO REAL;
	_pObjDesc		: POINTER TO STRING;

	_stEndDT		: ST_BACnet_DateTime;
	_nStartTimeDate	: UDINT; (* start time/date since 1900 in 100ms steps *)
	_nEndTimeDate	: UDINT; (* end time/date since 1900 in 100ms steps *)
END_VAR
VAR_TEMP
	_nTimeStamp		: UDINT;
END_VAR
(*

typedef struct _AnyType
{
      ULONG           nSize;
      BACnetDataTypes dataType;
      //... Data
}AnyType, *PAnyType;

enum BACnetLogRecordChoice
{
      logStatus,              // [0] BACnetLogStatus,
      booleanValue,           // [1] BOOL,
      realValue,              // [2] REAL,
      enumValue,              // [3] ENUMERATED, __ Optionally limited to 32 bits
      unsignedValue,          // [4] Unsigned, __ Optionally limited to 32 bits
      signedValue,            // [5] INTEGER, __ Optionally limited to 32 bits
      bitstringValue,         // [6] BIT STRING, __ Optionally limited to 32 bits
      nullValue,              // [7] NULL,
      failure,                // [8] Error,
      timeChange,             // [9] REAL,
      anyValue,               // [10] ABSTRACT_SYNTAX.&Type __ Optional
};

typedef struct _BACnetLogDatumList
{
      DWORD nEntrySize; // 0x80000000 -> next entry
      DWORD reserved;
      BACnetLogDatum listEntry;
}BACnetLogDatumList, *PBACnetLogDatumList;

typedef struct _BACnetLogDatum
{
      BACnetLogRecordChoice choice;
      union
      {
            DWORD logStatus; // BitString ... of type BACnetLogStatus
            BOOL booleanValue;
            FLOAT realValue;
            EnumerationValueType enumerationValue;
            ULONG unsignedValue;
            DWORD signedValue;
            DWORD bitstringValue;
            DWORD nullValue;
            BACnetError failure; 
            FLOAT timeChange;
            AnyType anyValue; // ABSTRACT-SYNTAX.&Type
      };
}BACnetLogDatum, *PBACnetLogDatum;


typedef struct _BACnetLogRecord
{
      ULONG validFields;
      BACnetDateTime timestamp;          // [0]
      DWORD statusFlags;                       // [2] optional
      BACnetLogDatumList logDatum;  // [1]
}BACnetLogRecord, *PBACnetLogRecord;

typedef struct _BACnetLogRecordList
{
      DWORD nEntrySize; // 0x80000000 -> next entry
      DWORD nSequence;  // "reserved"     -> Number of Sequence begins with 1
      BACnetLogRecord listEntry;
}BACnetLogRecordList, *PBACnetLogRecordList;

*)

(* ADS read *)
_fbReadProp(
	BACnetDevicePort	:= stAdsConn.nAmsPort,
	bExecute			:= ,
	sNetId				:= stAdsConn.sAmsNetId,
	ObjectType			:= F_BACnet_GetObjType(tObjectID),
	PropertyID			:= BACnetPropertyIdentifier_LogBuffer,
	DataType			:= BACnetDataType_LogRecordList,
	ObjectInstance		:= F_BACnet_GetObjInstance(tObjectID),
	ptrValue			:= ADR(stBACnet_AdsBuffer.arrData),
	nLenValue			:= SIZEOF(stBACnet_AdsBuffer.arrData),
	bDone				=> ,
	bBusy				=> ,
	bError				=> ,
	nErrID				=> ,
	nProcessedLen		=> );

_fbObjDesc(
	tObjectID	:= tObjectID,
	bAutoGet	:= FALSE,
	bGet		:= (_i = 1) AND (NOT _fbObjName.bBusy),
	stAdsConn	:= stAdsConn,
	bDone		=> ,
	bBusy		=> ,
	bError		=> ,
	nErrorId	=> ,
	sText		=> );

IF		(_fbObjDesc.bDone AND _fbObjDesc.sText = '')
	OR	_fbObjDesc.bError
THEN
	(* No description found, read name *)
	_fbObjName.bGet := TRUE;
ELSIF _fbObjDesc.bDone THEN
	(* OK, description found *)
	_pObjDesc := ADR(_fbObjDesc.sText);
END_IF

_fbObjName(
	tObjectID	:= tObjectID,
	bAutoGet	:= FALSE,
	bGet		:= ,
	stAdsConn	:= stAdsConn,
	bDone		=> ,
	bBusy		=> ,
	bError		=> ,
	nErrorId	=> ,
	sText		=> );

IF _fbObjName.bDone THEN
	(* OK, name found *)
	_pObjDesc := ADR(_fbObjName.sText);
END_IF
IF (NOT _fbObjName.bBusy) THEN
	_fbObjName.bGet := FALSE;
END_IF

(* trigger start event *)
_rtrigGet(CLK:= bGet, Q=> );

(* state machine *)
CASE _i OF

	0: (* Idle *)
		IF 		_rtrigGet.Q
			OR	(		(		(_nAdsReloadOld <> stAdsConn.nReload)
							OR	(_tObjectIDOld <> tObjectID)
						)
					AND	bAutoGet
				)
		THEN
			IF (NOT stAdsConn.bValid) THEN
				(* ADS connection not valid *)
				nErrorId := BACnet_ERR_INVALID_ADS_CONN;
			ELSIF (NOT stAdsConn.bServer AND NOT stAdsConn.bClient) THEN
				(* not a server nor a client *)
				nErrorId := BACnet_ERR_ADS_NoServerClient;
			ELSE
				_i := 1;
				nErrorId := BACnet_ERR_NO_ERROR;
				(* reset index *)
				_iEntry		:= 0;
				(* remind parameter *)
				_tObjectIDOld := tObjectID;
				_nAdsReloadOld := stAdsConn.nReload;
				(* clear object description index *)
				_pObjDesc := 0;
				(* reset start/end time/date *)
				_nStartTimeDate := 0;
				_nEndTimeDate := 0;
				_stEndDT := stEndTime;
			END_IF
			(* reset done flag *)
			bDone := FALSE;
		END_IF
		IF (NOT bGet) AND (NOT bAutoGet) THEN
			nErrorId := BACnet_ERR_NO_ERROR;
			bDone := FALSE;
		END_IF

	(* READ *)
	1: (* read object property data over ADS *)
		IF TestAndSet(stBACnet_AdsBuffer.bTestSet) THEN
			IF _fbReadProp.bExecute THEN
				IF _fbReadProp.bError THEN
					_i := 100;
					nErrorId := BACnet_ERR_ADS_Read;
					_fbReadProp.bExecute := FALSE;
				ELSIF (NOT _fbReadProp.bBusy) THEN
					_i := 2;
					_fbReadProp.bExecute := FALSE;
					(* prepare pointer *)
					_pAdsBuf := ADR(stBACnet_AdsBuffer.arrData);
					_pLbRecordList := _pAdsBuf;
					(* clear output data *)
					MEMSET(ADR(stLogBuffer.arrEntries), 0, SIZEOF(stLogBuffer.arrEntries));
					stLogBuffer.nCount := 0;
					stLogBuffer.sObjectDesc := '';
					_cbTotalBuf := 0;
					_iNextRecPos := 0;
					_nRecCount := 0;
					_nMaxSeq := 0;
				END_IF

			ELSIF (stBACnet_AdsBuffer.iLocked = 0) THEN
				_fbReadProp.bExecute := TRUE;
				(* lock global ADS buffer *)
				stBACnet_AdsBuffer.iLocked := SIZEOF(stBACnet_AdsBuffer.arrData);
			END_IF

			(* release temporary task lock *)
			stBACnet_AdsBuffer.bTestSet := FALSE;
		END_IF

	2: (* select record list entry *)
		REPEAT (* record list *)

			IF ((_pLbRecordList^.nEntrySize AND 16#7FFFFFFF) > 0) THEN

				(* check sequence order *)
				IF _nMaxSeq > _pLbRecordList^.nSequence THEN
					(* current sequence is lower then previous one - scan entries and sort *)
					FOR _iRec := 0 TO _nRecCount-1 DO
						IF _arrRecords[_iRec]^.nSequence > _pLbRecordList^.nSequence THEN
							(* found higher sequence no. - move *)
							_iNextRecPos := _iRec; (* remind insert position *)
							(* check free space *)
							IF (_nRecCount-1 < BACnet_MaxLogBufferEntries) THEN
								(* enough space at end of list - move *)
								MEMMOVE(	ADR(_arrRecords[_iRec+1]), (* one position up *)
											ADR(_arrRecords[_iRec]), (* free insert position *)
											(_nRecCount - _iRec)*SIZEOF(_arrRecords[0]) (* move all element behind insert position *)
								);
							END_IF
							EXIT; (* leave *)
						END_IF
					END_FOR
				ELSE
					(* remind sequence no. *)
					_nMaxSeq := _pLbRecordList^.nSequence;
				END_IF

				(* insert pointer to record entry *)
				_arrRecords[_iNextRecPos] := _pLbRecordList;
				(* select next free record position and count *)
				_iNextRecPos := _iNextRecPos + 1;
				_nRecCount := _nRecCount + 1;
			END_IF

			(* next record entry *)
			_NextLogRecord();

		UNTIL (		(NOT _bNextRecord) (* no more record entries *)
				OR	(_nRecCount >= (BACnet_MaxLogBufferEntries+1)) (* result buffer full *)
				OR	(_pLbRecordList >= (_pAdsBuf + stBACnet_AdsBuffer.iLocked)) (* ads buffer ending reached *)
			)
		END_REPEAT


		(* preset counter *)
		_iEntry := 0;
		(* scan sorted list *)
		FOR _iRec := 0 TO _nRecCount-1 DO
			(* take first date/time ... *)
			IF (_iRec = 0) THEN
				(* ...and merge with given start time *)
				_nStartTimeDate :=	F_BACnet_Get100msDate(F_BACnet_DateMerge(
										stStartTime.stDate,
										_arrRecords[_iRec]^.listEntry.timestamp.stDate)
									)
								+	F_BACnet_Get100msTime(F_BACnet_TimeMerge(
										stStartTime.stTime,
										_arrRecords[_iRec]^.listEntry.timestamp.stTime)
									);
				(* ...and merge with given end time *)
				IF F_BACnet_TimeUnspecified(_stEndDT.stTime) AND F_BACnet_DateUnspecified(_stEndDT.stDate) THEN
					_stEndDT := _arrRecords[_nRecCount-1]^.listEntry.timestamp;
				ELSE
					(* replace top down all placeholders with start time information *)
					IF _stEndDT.stTime.nHour = 16#FF THEN
						_stEndDT.stTime.nHour := _arrRecords[_iRec]^.listEntry.timestamp.stTime.nHour;
						IF _stEndDT.stTime.nMinute = 16#FF THEN
							_stEndDT.stTime.nMinute := _arrRecords[_iRec]^.listEntry.timestamp.stTime.nMinute;
							IF _stEndDT.stTime.nSecond = 16#FF THEN
								_stEndDT.stTime.nSecond := _arrRecords[_iRec]^.listEntry.timestamp.stTime.nSecond;
								IF _stEndDT.stTime.nHundredths = 16#FF THEN
									_stEndDT.stTime.nHundredths := _arrRecords[_iRec]^.listEntry.timestamp.stTime.nHundredths;
								END_IF
							END_IF
						END_IF
					END_IF
					(* replace time placeholder with maximum time values *)
					_stEndDT.stTime := F_BACnet_TimeMerge(_stEndDT.stTime, _stMaxTime);

					(* replace top down all placeholders with start date information *)
					IF _stEndDT.stDate.nYear = 16#FF THEN
						_stEndDT.stDate.nYear := _arrRecords[_iRec]^.listEntry.timestamp.stDate.nYear;
						IF _stEndDT.stDate.nMonth = 16#FF THEN
							_stEndDT.stDate.nMonth := _arrRecords[_iRec]^.listEntry.timestamp.stDate.nMonth;
							IF _stEndDT.stDate.nDay = 16#FF THEN
								_stEndDT.stDate.nDay := _arrRecords[_iRec]^.listEntry.timestamp.stDate.nDay;
								_stEndDT.stDate.nDayOfWeek := _arrRecords[_iRec]^.listEntry.timestamp.stDate.nDayOfWeek;
							END_IF
						END_IF
					END_IF
					(* replace date placeholder with maximum date values *)
					_stEndDT.stDate := F_BACnet_DateMerge(_stEndDT.stDate, _stMaxDate);
				END_IF

				(* calculate 100ms values for end time/date *)
				_nEndTimeDate := F_BACnet_Get100msTime(_stEndDT.stTime) + F_BACnet_Get100msDate(_stEndDT.stDate);
				IF _nEndTimeDate <= (		F_BACnet_Get100msTime(_arrRecords[_iRec]^.listEntry.timestamp.stTime)
										+	F_BACnet_Get100msDate(_arrRecords[_iRec]^.listEntry.timestamp.stDate)
									)
				THEN
					(* end time is lower than start time - set maximum value *)
					_nEndTimeDate := 	16#FFFFFFFF;
				END_IF
			END_IF

			(* initialize datum list pointer *)
			_pLrDatumList := ADR(_arrRecords[_iRec]^.listEntry.logDatum);

			REPEAT (* datum list *)

				(* check if local buffer is full *)
				IF _iEntry > BACnet_MaxLogBufferEntries THEN
					(* maximum entries reached --> finished *)
					_i := 4;
				ELSIF (_pLrDatumList^.nEntrySize AND 16#7FFFFFFF) > 0 THEN
					(* check time range *)
					_nTimeStamp :=	F_BACnet_Get100msDate(_arrRecords[_iRec]^.listEntry.timestamp.stDate)
								+	F_BACnet_Get100msTime(_arrRecords[_iRec]^.listEntry.timestamp.stTime);
					IF		(_nTimeStamp >= _nStartTimeDate) AND (_nTimeStamp <= _nEndTimeDate)
						AND	(_pLrDatumList^.listEntry.choice = BACnetLogRecordChoice_realValue)
					THEN
						(* append entry *)
						stLogBuffer.arrEntries[_iEntry].stDateTime := _arrRecords[_iRec]^.listEntry.timestamp;
						stLogBuffer.arrEntries[_iEntry].nTimeStamp := _nTimeStamp;
						_pReal := ADR(_pLrDatumList^.listEntry.nData);
						stLogBuffer.arrEntries[_iEntry].fValue := _pReal^;
						(* count up *)
						_iEntry := _iEntry + 1;
					END_IF
				END_IF

				(* next datum entry *)
				_NextLogDatum();

			UNTIL	(NOT _bNextDatum)
				OR	(_i <> 2)
			END_REPEAT

			(* exit if state changed *)
			IF _i <> 2 THEN EXIT; END_IF
		END_FOR
		_i := 4;


	4: (* wait on object description *)
		IF (NOT _fbObjDesc.bBusy) AND (NOT _fbObjName.bBusy) THEN
			(* set description *)
			IF _pObjDesc <> 0 THEN
				stLogBuffer.sObjectDesc := _pObjDesc^;
			ELSE
				stLogBuffer.sObjectDesc := F_BACnet_GetObjectIdString(tObjectID);
			END_IF
			(* set count *)
			stLogBuffer.nCount := _iEntry;
			stLogBuffer.nGet := stLogBuffer.nGet + 1;
			_i := 100;
		END_IF

	100: (* Done *)
		bDone := (nErrorId = BACnet_ERR_NO_ERROR);
		(* release ADS buffer *)
		stBACnet_AdsBuffer.iLocked := 0;
		(* go idle *)
		_i := 0;

END_CASE

(* set error flag *)
bError 	:= nErrorId > BACnet_ERR_NO_ERROR;
bBusy 	:= _i > 0;
END_FUNCTION_BLOCK
ACTION _NextLogDatum:
_bNextDatum := (_pLrDatumList^.nEntrySize AND 16#80000000) = 16#80000000;
_cbTmpSize := 	(_F_BACnet_AlignedSize(_pLrDatumList^.nEntrySize) AND 16#7FFFFFFF)
			+	SIZEOF(_pLrDatumList^.nEntrySize)
			+	SIZEOF(_pLrDatumList^.reserved);
_pLrDatumList := _pLrDatumList + _cbTmpSize;
END_ACTION
ACTION _NextLogRecord:
_bNextRecord := ((_pLbRecordList^.nEntrySize AND 16#80000000) = 16#80000000);
_cbTmpSize := _F_BACnet_AlignedSize(_pLbRecordList^.nEntrySize AND 16#7FFFFFFF) + SIZEOF(_pLbRecordList^.nEntrySize) + SIZEOF(_pLbRecordList^.nSequence);
_pLbRecordList	:= _pLbRecordList + _cbTmpSize;
_cbTotalBuf := _cbTotalBuf + _cbTmpSize;
END_ACTION

(* POU FB_BACnet_ObjectNameProperty, ST *)
FUNCTION_BLOCK FB_BACnet_ObjectNameProperty
VAR_INPUT
	tObjectID			: T_BACnet_ObjectIdentifier := 16#FFFFFFFF;
	bAutoGet			: BOOL:=TRUE; (* TRUE = get data from property when ADS connection OR object ID changed *)
	bGet				: BOOL; (* FALSE --> TRUE = get data from property *)
END_VAR
VAR_IN_OUT
	stAdsConn			: ST_BACnet_AdsConnection;
END_VAR
VAR_OUTPUT
	bDone				: BOOL;
	bBusy				: BOOL;
	bError				: BOOL;
	nErrorId			: UINT;
	sText				: T_MaxString; (* Object name *)
END_VAR
VAR
	_fbReadProp		: FB_BACnet_ReadProp;
	_i				: INT;
	_rtrigGetSet	: R_TRIG;
	_nAdsReloadOld	: USINT;
	_tObjectIDOld	: T_BACnet_ObjectIdentifier := 16#FFFFFFFF;
	_StringExtDecode: FB_BACnet_StringExtDecode;
END_VAR
(* ADS read *)
_fbReadProp(
	BACnetDevicePort	:= stAdsConn.nAmsPort,
	bExecute			:= ,
	sNetId				:= stAdsConn.sAmsNetId,
	ObjectType			:= F_BACnet_GetObjType(tObjectID),
	PropertyID			:= BACnetPropertyIdentifier_ObjectName,
	DataType			:= BACnetDataType_CharacterStringExt,
	ObjectInstance		:= F_BACnet_GetObjInstance(tObjectID),
	ptrValue			:= ADR(sText),
	nLenValue			:= SIZEOF(sText)-1,
	bDone				=> ,
	bBusy				=> ,
	bError				=> ,
	nErrID				=> ,
	nProcessedLen		=> );

(* trigger start event *)
_rtrigGetSet(CLK:= bGet, Q=> );

(* state machine *)
CASE _i OF

	0: (* Idle *)
		IF		(		(		_rtrigGetSet.Q
							OR	(_nAdsReloadOld <> stAdsConn.nReload)
							OR	(_tObjectIDOld <> tObjectID)
						)
					AND	bAutoGet
				)
			OR	_rtrigGetSet.Q
		THEN
			IF (NOT stAdsConn.bValid) THEN
				(* ADS connection not valid *)
				nErrorId := BACnet_ERR_INVALID_ADS_CONN;
			ELSIF (NOT stAdsConn.bServer AND NOT stAdsConn.bClient) THEN
				(* not a server nor a client *)
				nErrorId := BACnet_ERR_ADS_NoServerClient;
			ELSE
				nErrorId := BACnet_ERR_NO_ERROR;
				_i := 1;
				sText := '';
				(* remind ADS reload counter and parameter *)
				_nAdsReloadOld := stAdsConn.nReload;
				_tObjectIDOld := tObjectID;
			END_IF
			(* reset done flag *)
			bDone := FALSE;
		END_IF
		IF (NOT bGet) AND (NOT bAutoGet) THEN
			nErrorId := BACnet_ERR_NO_ERROR;
			bDone := FALSE;
		END_IF

	(* READ *)
	1: (* read object property data over ADS *)
		IF _fbReadProp.bExecute THEN
			IF _fbReadProp.bError THEN
				_i := 100;
				nErrorId := BACnet_ERR_ADS_Read;
				_fbReadProp.bExecute := FALSE;
			ELSIF (NOT _fbReadProp.bBusy) THEN
				_fbReadProp.bExecute := FALSE;
				(* decode property data *)
				_StringExtDecode(
					pChrStringExt	:= ADR(sText),
					cbOutSize		:= _fbReadProp.nProcessedLen,
					pOutString		:= ADR(sText),
					bValid			=> ,
					bOverflow		=> ,
					nLength			=> ,
					eSrcEncoding	=> );
				(* check overflow flag *)
				IF _StringExtDecode.bOverflow THEN
					nErrorId := BACnet_ERR_ADS_BufferSize;
				END_IF
				(* DONE *)
				_i := 100;
			END_IF
		ELSE
			_fbReadProp.bExecute := TRUE;
		END_IF

	100: (* Done *)
		bDone := (nErrorId = BACnet_ERR_NO_ERROR);
		_i := 0;

END_CASE

(* set error flag *)
bError 	:= nErrorId > BACnet_ERR_NO_ERROR;
bBusy 	:= _i > 0;
END_FUNCTION_BLOCK

(* POU FB_BACnet_Loop, ST *)
FUNCTION_BLOCK FB_BACnet_Loop
VAR_INPUT
	fAccLimit		: REAL := 0.0; (* Setpoint acceleration limit positive and negative [1/s] *)
END_VAR
VAR_IN_OUT
	Device			: FB_BACnet_Device;
END_VAR
VAR_OUTPUT
	bReady			: BOOL;
	fSetPoint		: REAL;
	fControlledValue: REAL;
	fPresentValue	: REAL;
	fPropBand		: REAL; (* controller output in range of -100...100% in relation to Min.-/Max.-output *)
	bOverridden		: BOOL;
	bOutOfService	: BOOL;
	bFault			: BOOL;
	bInAlarm		: BOOL;
	bOpenLoop		: BOOL;
	bCommFailure	: BOOL;
	bOtherFault		: BOOL;
	bError			: BOOL;
	nErrorId		: UINT;
	eMode			: E_BACNETLOOPMODE; (* mode is detected by the unit of property Integral_Constant and Derivative_Constant (Time_seconds = BACnetLoopMode_Standard) *)
END_VAR
VAR
	_ControlledVariableValue AT%I*: REAL;	(* ~(BACnet_ControlledVariableValue :		: )
												(BACnet_ObjectType				: LOOP	: )	*)
	_Setpoint AT%I*:REAL;					(* ~(BACnet_Setpoint				:		: )	*)
	_ProportionalConstant AT%I*:REAL;		(* ~(BACnet_ProportionalConstant	:		: )	*)
	_IntegralConstant AT%I*:REAL;			(* ~(BACnet_IntegralConstant	 	:		: )	*)
	_DerivativeConstant AT%I*:REAL;			(* ~(BACnet_DerivativeConstant	 	:		: )	*)
	_MaximumOutput AT%I*:REAL;				(* ~(BACnet_MaximumOutput			:		: )	*)
	_MinimumOutput AT%I*:REAL;				(* ~(BACnet_MinimumOutput			:		: )	*)
	_Bias AT%I*:REAL;						(* ~(BACnet_Bias					:		: )	*)
	_PresentValueI AT%I*: REAL; 			(* ~(BACnet_PresentValue 			: 		: )	*)
	_StatusFlags AT%I*: WORD; 				(* ~(BACnet_StatusFlags 			: 		: )	*)
	_Reliability AT%I*: E_BACNETRELIABILITY;(* ~(BACNET_RELIABILITY 			:		: )	*)
	_ControlAction AT%I*:E_BACNETACTION;	(* ~(BACNET_ACTION				 	:		: )	*)
	_PropConstantUnits AT%I*:E_BACNETUNIT;	(* ~(BACnet_ProportionalConstantUnits:	Other_no_units	: WRITEPROTECT) *)
	_IntegralConstUnits AT%I*:E_BACNETUNIT;	(* ~(BACnet_IntegralConstantUnits	:	Other_no_units	: WRITEPROTECT) *)
	_DerivativeConstUnits AT%I*:E_BACNETUNIT;(*~(BACnet_DerivativeConstantUnits	:	Other_no_units	: WRITEPROTECT) *)
	_PresentValueQ AT%Q*: REAL;				(* ~(BACnet_PresentValue	 		:		: )	*)
	_StatusFlagsBits : ST_BACnet_StatusFlags;

	_sysTime	: GETCPUCOUNTER;
	_Time		: T_LARGE_INTEGER;
	_TimeOld	: T_LARGE_INTEGER;
	_cycleTime	: REAL;
	_PidControl : FB_BACnet_PidControl;
	_fbAccLimit : FB_BACnet_AccLimit;

	_nUpdateCount : UDINT := 0;
END_VAR
(* update server device *)
IF (Device._nUpdateCount = _nUpdateCount) THEN
	Device();
END_IF
(* remind current number of update counter *)
_nUpdateCount := Device._nUpdateCount;

(* determine cycle time *)
_TimeOld := _Time;
_sysTime(cpuCntLoDW=> _Time.dwLowPart, cpuCntHiDW=> _Time.dwHighPart);
_cycleTime := _F_BACnet_SysTimeDiff(In1:=_Time, In2:=_TimeOld);

(* check BitString format of StatusFlags --> if StatusFlags are less than 4, object isn't linked correctly *)
IF (_StatusFlags < 4) THEN
	(* wrong mapping *)
	nErrorId := BACnet_ERR_WRONG_MAPPING;
	bReady := FALSE;

ELSIF Device.bOperational THEN
	(* ready state *)
	bReady := TRUE;
	nErrorId := BACnet_ERR_NO_ERROR;

	(* decode status flags *)
	_StatusFlagsBits := F_BACnet_StatusFlags(_StatusFlags);

	(* copy states to output *)
	bOverridden := _StatusFlagsBits.overridden;
	bOutOfService := _StatusFlagsBits.out_of_service;
	bFault := _StatusFlagsBits.fault;
	bInAlarm := _StatusFlagsBits.in_alarm;
	bOpenLoop := (_Reliability = BACnetReliability_open_loop);
	bCommFailure := (_Reliability = BACnetReliability_communication_failure);
	bOtherFault := (_Reliability = BACnetReliability_unreliable_other);

	(* check PID mode *)
	IF		((_IntegralConstUnits = BACnetUnit_Time_seconds OR _IntegralConstUnits = 0) AND _DerivativeConstUnits = BACnetUnit_Time_seconds)
		AND	((_DerivativeConstUnits = BACnetUnit_Time_seconds OR _DerivativeConstUnits = 0) AND _IntegralConstUnits = BACnetUnit_Time_seconds)
		AND (_PropConstantUnits = BACnetUnit_Other_no_units)
	THEN
		(* both are time_seconds *)
		eMode := BACnetLoopMode_Standard;
	ELSIF	(_IntegralConstUnits <> BACnetUnit_Time_seconds)
		AND	(_DerivativeConstUnits <> BACnetUnit_Time_seconds)
		AND (_PropConstantUnits = BACnetUnit_Other_no_units)
		(* both are not time_seconds *)
	THEN
		eMode := BACnetLoopMode_Ideal;
	ELSE
		(* unknown settings - stop controller *)
		eMode := BACnetLoopMode_None;
	END_IF

	(* check reliability and mode *)
	IF		(_Reliability <> BACnetReliability_no_fault_detected)
		OR	(eMode = BACnetLoopMode_None)
	THEN
		_PidControl.bReset			:= TRUE;

	(* is set out of service? *)
	ELSIF _StatusFlagsBits.out_of_service THEN
		_PidControl.bReset			:= TRUE;

	(* decide the control action (direct or reverse) *)
	ELSIF _ControlAction = BACnetAction_direct THEN
		_PidControl.bReset			:= FALSE;
		_PidControl.fPresentValue	:= _ControlledVariableValue;
		_PidControl.fSetpoint		:= _Setpoint;

	ELSIF _ControlAction = BACnetAction_reverse THEN
		_PidControl.bReset			:= FALSE;
		_PidControl.fPresentValue	:= _Setpoint;
		_PidControl.fSetpoint		:= _ControlledVariableValue;

	ELSE
		(* unknown action *)
		_PidControl.bReset			:= TRUE;
	END_IF

	(* set parameter depending on mode *)
	CASE eMode OF
		BACnetLoopMode_Ideal:
			_PidControl.fKp := _ProportionalConstant;
			_PidControl.fKi	:= _IntegralConstant;
			_PidControl.fKd	:= _DerivativeConstant;
		BACnetLoopMode_Standard:
			(* Kp = Kp *)
			_PidControl.fKp := _ProportionalConstant;
			(* Ki = Kp / Ti *)
			IF (_IntegralConstant <> 0.0) THEN
				_PidControl.fKi	:= _ProportionalConstant / _IntegralConstant;
			ELSE
				_PidControl.fKi	:= 0.0;
			END_IF
			(* Kd = Kp * Td *)
			_PidControl.fKd	:= _ProportionalConstant * _DerivativeConstant;
	END_CASE

	(* call PID control function block *)
	_PidControl(
		fCtrlCycleTime	:= _cycleTime,
		fBias			:= _Bias,
		fTp				:= -1.0,
		fMaxOutput		:= _MaximumOutput,
		fMinOutput		:= _MinimumOutput,
		nErrorStatus	=>
	);
	_fbAccLimit.X := _PidControl.fY;

	(* set other outputs *)
	fSetPoint := _Setpoint;
	fPresentValue := _PresentValueI;
	fControlledValue := _ControlledVariableValue;
ELSE
	(* server device not ready, reset local ready also *)
	bReady := FALSE;
	nErrorId := BACnet_ERR_OPERATIONAL;
END_IF

(* limit present value *)
_fbAccLimit(X:= , Amax:= fAccLimit, Tcycle:= _cycleTime, Y=> _PresentValueQ, A=> );

(* calculate proportional band *)
IF (_MaximumOutput > 0.0) AND (_MinimumOutput >= 0.0) THEN
	fPropBand := ((_PresentValueQ - _MinimumOutput) / (_MaximumOutput - _MinimumOutput)) * 100.0;
ELSIF (_MaximumOutput <= 0.0) AND (_MinimumOutput < 0.0) THEN
	fPropBand := ((_PresentValueQ - _MaximumOutput) / (_MaximumOutput - _MinimumOutput)) * 100.0;
ELSIF (_PresentValueQ > 0.0) AND (_MaximumOutput > 0.0) THEN
	fPropBand := (_PresentValueQ / _MaximumOutput) * 100.0;
ELSIF (_PresentValueQ < 0.0) AND (_MinimumOutput < 0.0) THEN
	fPropBand := (_PresentValueQ / _MinimumOutput) * -100.0;
ELSE
	fPropBand := 0.0;
END_IF

(* set error flag *)
bError := (nErrorId <> BACnet_ERR_NO_ERROR);
END_FUNCTION_BLOCK

(* POU FB_BACnet_PidControl, ST *)
FUNCTION_BLOCK FB_BACnet_PidControl
VAR_INPUT
	(* controller input  *)
	fSetpoint				: REAL;	(* setpoint value *)
	fPresentValue			: REAL;	(* actual value *)
	(* reset flag *)
	bReset					: BOOL;
	(* controller values *)
	fCtrlCycleTime			: REAL; (* controller cycle time in seconds [s] *)

	fBias					: REAL; (* bias also active when reset is set to 1 *)
	fKp						: REAL;	(* proportional gain Kp	(P) *)
	fKi						: REAL; (* integral gain Ki (I) *)
	fKd						: REAL;	(* derivative gain Kd (D) *)
	fTp						: REAL := -1.0;	(* damping time Tp (PT1) [s] (fTp < 0 --> Tp = Kd / 10) *)

	(* maximum ratings *)
	fMaxOutput				: REAL;
	fMinOutput				: REAL;
END_VAR
VAR_OUTPUT
	fY						: REAL; (* controller output command *)
	nErrorStatus			: UINT; (* controller error output (0: no error; >0:error) *)
END_VAR
VAR
	(* Internal Variable *)
	_fE		: REAL;
	_fEOld	: REAL;
	_fYp	: REAL;
	_fYi	: REAL;
	_fYd	: REAL;
	_fbYd	: FB_BACnet_PT1;
END_VAR
(* preset error number *)
nErrorStatus	:= BACnet_ERR_NO_ERROR;

(* check cycle time parameter: (CycleTime > 0) *)
IF (fCtrlCycleTime <= 0.0) THEN
	nErrorStatus := BACnet_ERR_INVALID_CYCLETIME;
	bReset := TRUE;
END_IF;

(* check controller parameters: (Kp, Ki, Kd >= 0) *)
IF ((fKp < 0.0) OR (fKi < 0.0) OR (fKd < 0.0)) THEN
	nErrorStatus := BACnet_ERR_INVALID_PARAMETER;
	bReset := TRUE;
END_IF;

(* controller reset *)
IF bReset THEN
	(* reset internal and external variables *)
	_fEOld	:= 0.0;
	fY		:= MAX(MIN(fBias, fMaxOutput), fMinOutput);
	_fYi	:= 0.0;
	_fbYd(X:= 0.0, T:= 0.0, Y=> );
	RETURN;
END_IF

(* 3. save old variable *)
_fEOld := _fE;

(* 4. set error/deviation input *)
_fE := fSetpoint - fPresentValue;

(* 5. YP-part *)
_fYp := fKp * _fE;

(* 6. YI-part *)
IF (fKi = 0.0) THEN
	_fYi	:= 0.0;
ELSE
	_fYi := _fYi + (fKi * fCtrlCycleTime * _fE);
END_IF
IF (_fYi > fMaxOutput) THEN
	(* limit wind up positive *)
	_fYi := fMaxOutput;
ELSIF (_fYi < fMinOutput) THEN
	(* limit wind up negative *)
	_fYi := fMinOutput;
END_IF

(* 7. YD-part *)
IF (fTp < 0.0) THEN
	fTp := fKd / 10.0;
END_IF
_fYd := fKd * (_fE - _fEOld) / fCtrlCycleTime;
_fbYd(X:= _fYd, T:= fTp, Tcycle:= fCtrlCycleTime, Y=> );

(* 8. Ysum = YP + YI + YD + Bias and output *)
fY := _fYp + _fYi + _fbYd.Y + fBias;
fY := MAX(MIN(fY, fMaxOutput), fMinOutput);
END_FUNCTION_BLOCK

(* POU FB_BACnet_Loop_DRV, ST *)
FUNCTION_BLOCK FB_BACnet_Loop_DRV
VAR_IN_OUT
	Device	: FB_BACnet_Device;
END_VAR
VAR_OUTPUT
	bReady				: BOOL;
	fSetPoint			: REAL;
	fControlledValue	: REAL;
	fPresentValue		: REAL;
	bOverridden			: BOOL;
	bOutOfService		: BOOL;
	bFault				: BOOL;
	bInAlarm			: BOOL;
	bError				: BOOL;
	nErrorId			: UINT;
END_VAR
VAR
	_ControlledVariableValue AT%I*: REAL;	(* ~(BACnet_ControlledVariableValue :		: )
												(BACnet_ObjectType				: LOOP	: )
												(BACnet_EnableInternalLoopCtrl	: TRUE	: NOLINK,ENABLE) *)
	_Setpoint AT%I*:REAL;					(* ~(BACnet_Setpoint				:		: )	*)
	_PresentValue AT%I*: REAL; 				(* ~(BACnet_PresentValue 			: 		: )	*)
	_ObjectId AT%I*: DWORD;					(* ~(BACnet_ObjectIdentifier		:		: LINK) *)
	_StatusFlags AT%I*: WORD; 				(* ~(BACnet_StatusFlags 			: 		: )	*)
	_StatusFlagsBits : ST_BACnet_StatusFlags;
	_nUpdateCount : UDINT := 0;
END_VAR
(* update server device *)
IF (Device._nUpdateCount = _nUpdateCount) THEN
	Device();
END_IF
(* remind current number of update counter *)
_nUpdateCount := Device._nUpdateCount;

(* check BitString format of StatusFlags --> if StatusFlags are less than 4, object isn't linked correctly *)
IF (_StatusFlags < 4) THEN
	(* wrong mapping *)
	nErrorId := BACnet_ERR_WRONG_MAPPING;
	bReady := FALSE;

ELSIF Device.bOperational THEN
	(* ready state *)
	bReady := TRUE;
	nErrorId := BACnet_ERR_NO_ERROR;

	(* decode status flags *)
	_StatusFlagsBits := F_BACnet_StatusFlags(_StatusFlags);

	(* copy states to output *)
	bOverridden := _StatusFlagsBits.overridden;
	bOutOfService := _StatusFlagsBits.out_of_service;
	bFault := _StatusFlagsBits.fault;
	bInAlarm := _StatusFlagsBits.in_alarm;

	(* set other outputs *)
	fSetPoint := _Setpoint;
	fPresentValue := _PresentValue;
	fControlledValue := _ControlledVariableValue;
ELSE
	(* server device not ready, reset local ready also *)
	bReady := FALSE;
	nErrorId := BACnet_ERR_OPERATIONAL;
END_IF
(* set error flag *)
bError := (nErrorId <> BACnet_ERR_NO_ERROR);
END_FUNCTION_BLOCK

(* POU FB_BACnet_Loop_DRV_EX, ST *)
FUNCTION_BLOCK FB_BACnet_Loop_DRV_EX
VAR_IN_OUT
	Device	: FB_BACnet_Device;
END_VAR
VAR_OUTPUT
	bReady				: BOOL;
	fSetPoint			: REAL;
	fControlledValue	: REAL;
	fPresentValue		: REAL;
	fPropBand			: REAL; (* controller output in range of -100...100% in relation to Min.-/Max.-output *)
	bOverridden			: BOOL;
	bOutOfService		: BOOL;
	bFault				: BOOL;
	bInAlarm			: BOOL;
	bOpenLoop			: BOOL;
	bCommFailure		: BOOL;
	bOtherFault			: BOOL;
	eEventState			: E_BACNETEVENTSTATE;
	bAckedTrans_ToOffNormal : BOOL;
	bAckedTrans_ToFault		: BOOL;
	bAckedTrans_ToNormal	: BOOL;
	tObjectID			: T_BACnet_ObjectIdentifier := 16#FFFFFFFF;
	bError				: BOOL;
	nErrorId			: UINT;
END_VAR
VAR
	_ControlledVariableValue AT%I*: REAL;	(* ~(BACnet_ControlledVariableValue :		: )
												(BACnet_ObjectType				: LOOP	: )
												(BACnet_EnableInternalLoopCtrl	: TRUE	: NOLINK,ENABLE) *)
	_Setpoint AT%I*:REAL;					(* ~(BACnet_Setpoint				:		: )	*)
	_MaximumOutput AT%I*:REAL;				(* ~(BACnet_MaximumOutput			:		: )	*)
	_MinimumOutput AT%I*:REAL;				(* ~(BACnet_MinimumOutput			:		: )	*)
	_PresentValue AT%I*: REAL; 				(* ~(BACnet_PresentValue 			: 		: )	*)
	_ObjectId AT%I*: DWORD;					(* ~(BACnet_ObjectIdentifier		:		: LINK) *)
	_StatusFlags AT%I*: WORD; 				(* ~(BACnet_StatusFlags 			: 		: )	*)
	_AckedTransitions AT%I*:WORD;			(* ~(BACnet_AckedTransitions		:		: ) *)
	_EventState AT%I*: WORD; 				(* ~(BACnet_EventState 				:		: )	*)
	_Reliability AT%I*: E_BACNETRELIABILITY;(* ~(BACNET_RELIABILITY 			:		: )	*)
	_StatusFlagsBits : ST_BACnet_StatusFlags;
	_AckedTransBits : ST_BACnet_EventTransitionBits;
	_nUpdateCount : UDINT := 0;
END_VAR
(* update server device *)
IF (Device._nUpdateCount = _nUpdateCount) THEN
	Device();
END_IF
(* remind current number of update counter *)
_nUpdateCount := Device._nUpdateCount;

(* check BitString format of StatusFlags --> if StatusFlags are less than 4, object isn't linked correctly *)
IF (F_BACnet_GetObjType(_ObjectId) <> BACnetObjectType_Loop) THEN
	(* wrong mapping / invalid object ID *)
	IF _ObjectId = 0 THEN
		nErrorId := BACnet_ERR_WRONG_MAPPING;
	ELSE
		nErrorId := BACnet_ERR_INVALID_OBJECTID;
	END_IF
	bReady := FALSE;
	tObjectID := 16#FFFFFFFF;

ELSIF (_StatusFlags < 4) THEN
	(* wrong mapping *)
	nErrorId := BACnet_ERR_WRONG_MAPPING;
	bReady := FALSE;

ELSIF Device.bOperational THEN
	(* ready state *)
	bReady := TRUE;
	nErrorId := BACnet_ERR_NO_ERROR;

	(* decode status flags *)
	_StatusFlagsBits := F_BACnet_StatusFlags(_StatusFlags);
	_AckedTransBits	:= F_BACnet_EventTransitionFlags(_AckedTransitions);

	(* copy states to output *)
	bOverridden := _StatusFlagsBits.overridden;
	bOutOfService := _StatusFlagsBits.out_of_service;
	bFault := _StatusFlagsBits.fault;
	bInAlarm := _StatusFlagsBits.in_alarm;
	bOpenLoop := (_Reliability = BACnetReliability_open_loop);
	bCommFailure := (_Reliability = BACnetReliability_communication_failure);
	bOtherFault := (_Reliability = BACnetReliability_unreliable_other);
	bAckedTrans_ToOffNormal := _AckedTransBits.to_offnormal;
	bAckedTrans_ToFault := _AckedTransBits.to_fault;
	bAckedTrans_ToNormal := _AckedTransBits.to_normal;
	tObjectID := _ObjectId;
	eEventState := _EventState;

	(* calculate proportional band *)
	IF (_MaximumOutput > 0.0) AND (_MinimumOutput >= 0.0) THEN
		fPropBand := ((_PresentValue - _MinimumOutput) / (_MaximumOutput - _MinimumOutput)) * 100.0;
	ELSIF (_MaximumOutput <= 0.0) AND (_MinimumOutput < 0.0) THEN
		fPropBand := ((_PresentValue - _MaximumOutput) / (_MaximumOutput - _MinimumOutput)) * 100.0;
	ELSIF (_PresentValue > 0.0) AND (_MaximumOutput > 0.0) THEN
		fPropBand := (_PresentValue / _MaximumOutput) * 100.0;
	ELSIF (_PresentValue < 0.0) AND (_MinimumOutput < 0.0) THEN
		fPropBand := (_PresentValue / _MinimumOutput) * -100.0;
	ELSE
		fPropBand := 0.0;
	END_IF

	(* set other outputs *)
	fSetPoint := _Setpoint;
	fPresentValue := _PresentValue;
	fControlledValue := _ControlledVariableValue;
ELSE
	(* server device not ready, reset local ready also *)
	bReady := FALSE;
	nErrorId := BACnet_ERR_OPERATIONAL;
END_IF
(* set error flag *)
bError := (nErrorId <> BACnet_ERR_NO_ERROR);
END_FUNCTION_BLOCK

(* POU FB_BACnet_Loop_EX, ST *)
FUNCTION_BLOCK FB_BACnet_Loop_EX
VAR_INPUT
	bAutoTuning			: BOOL; (* Start autotuning of PID controller *)
	tTuningTimeout		: TIME := T#15m; (* Maximum runtime of tuning procedure [ms] *)
	eTuningMode			: E_BACNETPIDTUNINGMODE := BACnetPIDTuningMode_PI; (* optimize default PI controller *)
	fAccLimit			: REAL := 0.0; (* Setpoint acceleration limit positive and negative [1/s] *)
END_VAR
VAR_IN_OUT
	Device				: FB_BACnet_Device;
END_VAR
VAR_OUTPUT
	bReady				: BOOL;
	bTuningActive		: BOOL;
	bTuningWaitPV		: BOOL;
	bTuningWaitCV		: BOOL;
	bTuningDone			: BOOL;
	bTuningAborted		: BOOL;
	fSetPoint			: REAL;
	fControlledValue	: REAL;
	fPresentValue		: REAL;
	fPropBand			: REAL; (* controller output in range of -100...100% in relation to Min.-/Max.-output *)
	bOverridden			: BOOL;
	bOutOfService		: BOOL;
	bFault				: BOOL;
	bInAlarm			: BOOL;
	bOpenLoop			: BOOL;
	bCommFailure		: BOOL;
	bOtherFault			: BOOL;
	eEventState			: E_BACNETEVENTSTATE;
	bAckedTrans_ToOffNormal : BOOL;
	bAckedTrans_ToFault		: BOOL;
	bAckedTrans_ToNormal	: BOOL;
	tObjectID			: T_BACnet_ObjectIdentifier := 16#FFFFFFFF;
	bError				: BOOL;
	nErrorId			: UINT;
	eMode				: E_BACNETLOOPMODE; (* mode is detected by the unit of property Integral_Constant and Derivative_Constant (Time_seconds = BACnetLoopMode_Standard) *)
END_VAR
VAR
	_ControlledVariableValue AT%I*: REAL;	(* ~(BACnet_ControlledVariableValue :		: )
												(BACnet_ObjectType				: LOOP	: )	*)
	_Setpoint AT%I*:REAL;					(* ~(BACnet_Setpoint				:		: )	*)
	_ProportionalConstant AT%I*:REAL;		(* ~(BACnet_ProportionalConstant	:		: )	*)
	_IntegralConstant AT%I*:REAL;			(* ~(BACnet_IntegralConstant	 	:		: )	*)
	_DerivativeConstant AT%I*:REAL;			(* ~(BACnet_DerivativeConstant	 	:		: )	*)
	_MaximumOutput AT%I*:REAL;				(* ~(BACnet_MaximumOutput			:		: )	*)
	_MinimumOutput AT%I*:REAL;				(* ~(BACnet_MinimumOutput			:		: )	*)
	_Bias AT%I*:REAL;						(* ~(BACnet_Bias					:		: )	*)
	_PresentValueI AT%I*: REAL; 			(* ~(BACnet_PresentValue 			: 		: )	*)
	_Deadband AT%I*: REAL; 					(* ~(BACnet_Deadband	 			: 		: )	*)
	_ObjectId AT%I*: DWORD;					(* ~(BACnet_ObjectIdentifier		:		: LINK) *)
	_StatusFlags AT%I*: WORD; 				(* ~(BACnet_StatusFlags 			: 		: )	*)
	_AckedTransitions AT%I*:WORD;			(* ~(BACnet_AckedTransitions		:		: ) *)
	_EventState AT%I*: WORD; 				(* ~(BACnet_EventState 				:		: )	*)
	_Reliability AT%I*: E_BACNETRELIABILITY;(* ~(BACNET_RELIABILITY 			:		: )	*)
	_ControlAction AT%I*:E_BACNETACTION;	(* ~(BACNET_ACTION				 	:		: )	*)
	_PropConstantUnits AT%I*:E_BACNETUNIT;	(* ~(BACnet_ProportionalConstantUnits:	Other_no_units	: WRITEPROTECT) *)
	_IntegralConstUnits AT%I*:E_BACNETUNIT;	(* ~(BACnet_IntegralConstantUnits	:	Other_no_units	: WRITEPROTECT) *)
	_DerivativeConstUnits AT%I*:E_BACNETUNIT;(*~(BACnet_DerivativeConstantUnits	:	Other_no_units	: WRITEPROTECT) *)
	_PresentValueQ AT%Q*: REAL;				(* ~(BACnet_PresentValue	 		:		: )	*)
	_AckedTransBits : ST_BACnet_EventTransitionBits;
	_StatusFlagsBits : ST_BACnet_StatusFlags;

	_sysTime	: GETCPUCOUNTER;
	_Time		: T_LARGE_INTEGER;
	_TimeOld	: T_LARGE_INTEGER;
	_cycleTime	: REAL;
	_PidControl : FB_BACnet_PidControl;
	_AutoTuning : _FB_BACnet_PidTune;
	_iTuning	: INT;
	_WriteProp	: FB_BACnet_WriteProp;
	_fbAccLimit : FB_BACnet_AccLimit;
	_nUpdateCount : UDINT := 0;

	_fTuneKp	: REAL;
	_fTuneKi	: REAL;
	_fTuneKd	: REAL;

END_VAR
(* update server device *)
IF (Device._nUpdateCount = _nUpdateCount) THEN
	Device();
END_IF
(* remind current number of update counter *)
_nUpdateCount := Device._nUpdateCount;

(* determine cycle time *)
_TimeOld := _Time;
_sysTime(cpuCntLoDW=> _Time.dwLowPart, cpuCntHiDW=> _Time.dwHighPart);
_cycleTime := _F_BACnet_SysTimeDiff(In1:=_Time, In2:=_TimeOld);

(* check BitString format of StatusFlags --> if StatusFlags are less than 4, object isn't linked correctly *)
IF (F_BACnet_GetObjType(_ObjectId) <> BACnetObjectType_Loop) THEN
	(* wrong mapping / invalid object ID *)
	IF _ObjectId = 0 THEN
		nErrorId := BACnet_ERR_WRONG_MAPPING;
	ELSE
		nErrorId := BACnet_ERR_INVALID_OBJECTID;
	END_IF
	bReady := FALSE;
	tObjectID := 16#FFFFFFFF;

ELSIF (_StatusFlags < 4) THEN
	(* wrong mapping *)
	nErrorId := BACnet_ERR_WRONG_MAPPING;
	bReady := FALSE;

ELSIF Device.bOperational THEN
	(* ready state *)
	bReady := TRUE;
	nErrorId := BACnet_ERR_NO_ERROR;

	(* decode status flags *)
	_StatusFlagsBits := F_BACnet_StatusFlags(_StatusFlags);
	_AckedTransBits	:= F_BACnet_EventTransitionFlags(_AckedTransitions);

	(* copy states to output *)
	bOverridden := _StatusFlagsBits.overridden;
	bOutOfService := _StatusFlagsBits.out_of_service;
	bFault := _StatusFlagsBits.fault;
	bInAlarm := _StatusFlagsBits.in_alarm;
	bOpenLoop := (_Reliability = BACnetReliability_open_loop);
	bCommFailure := (_Reliability = BACnetReliability_communication_failure);
	bOtherFault := (_Reliability = BACnetReliability_unreliable_other);
	bAckedTrans_ToOffNormal := _AckedTransBits.to_offnormal;
	bAckedTrans_ToFault := _AckedTransBits.to_fault;
	bAckedTrans_ToNormal := _AckedTransBits.to_normal;
	tObjectID := _ObjectId;
	eEventState := _EventState;

	(* check PID mode *)
	IF		((_IntegralConstUnits = BACnetUnit_Time_seconds OR _IntegralConstUnits = 0) AND _DerivativeConstUnits = BACnetUnit_Time_seconds)
		AND	((_DerivativeConstUnits = BACnetUnit_Time_seconds OR _DerivativeConstUnits = 0) AND _IntegralConstUnits = BACnetUnit_Time_seconds)
		AND (_PropConstantUnits = BACnetUnit_Other_no_units)
	THEN
		(* both are time_seconds *)
		eMode := BACnetLoopMode_Standard;
	ELSIF	(_IntegralConstUnits <> BACnetUnit_Time_seconds)
		AND	(_DerivativeConstUnits <> BACnetUnit_Time_seconds)
		AND (_PropConstantUnits = BACnetUnit_Other_no_units)
		(* both are not time_seconds *)
	THEN
		eMode := BACnetLoopMode_Ideal;
	ELSE
		(* unknown settings - stop controller *)
		eMode := BACnetLoopMode_None;
	END_IF

	(* check if auto tuning is active *)
	IF bTuningActive THEN
		_PidControl.bReset			:= TRUE;

	(* check reliability and mode *)
	ELSIF		(_Reliability <> BACnetReliability_no_fault_detected)
		OR	(eMode = BACnetLoopMode_None)
	THEN
		_PidControl.bReset			:= TRUE;

	(* is set out of service? *)
	ELSIF _StatusFlagsBits.out_of_service THEN
		_PidControl.bReset			:= TRUE;

	(* decide the control action (direct or reverse) *)
	ELSIF _ControlAction = BACnetAction_direct THEN
		_PidControl.bReset			:= FALSE;
		_PidControl.fPresentValue	:= _ControlledVariableValue;
		_PidControl.fSetpoint		:= _Setpoint;

	ELSIF _ControlAction = BACnetAction_reverse THEN
		_PidControl.bReset			:= FALSE;
		_PidControl.fPresentValue	:= _Setpoint;
		_PidControl.fSetpoint		:= _ControlledVariableValue;

	ELSE
		(* unknown action *)
		_PidControl.bReset			:= TRUE;
	END_IF

	(* set parameter depending on mode *)
	CASE eMode OF
		BACnetLoopMode_Ideal:
			_PidControl.fKp := _ProportionalConstant;
			_PidControl.fKi	:= _IntegralConstant;
			_PidControl.fKd	:= _DerivativeConstant;
		BACnetLoopMode_Standard:
			(* Kp = Kp *)
			_PidControl.fKp := _ProportionalConstant;
			(* Ki = Kp / Ti *)
			IF (_IntegralConstant <> 0.0) THEN
				_PidControl.fKi	:= _ProportionalConstant / _IntegralConstant;
			ELSE
				_PidControl.fKi	:= 0.0;
			END_IF
			(* Kd = Kp * Td *)
			_PidControl.fKd	:= _ProportionalConstant * _DerivativeConstant;
	END_CASE

	(* call PID control function block *)
	_PidControl(
		fCtrlCycleTime	:= _cycleTime,
		fBias			:= _Bias,
		fTp				:= -1.0,
		fMaxOutput		:= _MaximumOutput,
		fMinOutput		:= _MinimumOutput,
		nErrorStatus	=>
	);
	IF (_iTuning < 10) THEN
		_fbAccLimit.X := _PidControl.fY;
	END_IF

	(* set other outputs *)
	fSetPoint := _Setpoint;
	fPresentValue := _PresentValueI;
	fControlledValue := _ControlledVariableValue;
ELSE
	(* server device not ready, reset local ready also *)
	bReady := FALSE;
	nErrorId := BACnet_ERR_OPERATIONAL;
END_IF

(* write controller settings *)
_WriteProp.BACnetDevicePort:= Device.stAdsConn.nAmsPort;
_WriteProp.sNetId		:= Device.stAdsConn.sAmsNetId;
_WriteProp.ObjectType	:= BACnetObjectType_Loop;
_WriteProp.ObjectInstance:= F_BACnet_GetObjInstance(_ObjectId);

(* Autotuning function *)
CASE _iTuning OF
	0: (* Idle *)
		IF		bReady						(* object ready *)
			AND	(NOT _PidControl.bReset)	(* PID controller ready *)
			AND (tTuningTimeout > t#0ms)	(* timeout valid *)
			AND bAutoTuning					(* start flag *)
		THEN
			_iTuning := 5;
		END_IF
		_AutoTuning.bStart := FALSE;

	5:
		(* present_value low *)
		IF (_PresentValueI <= ((_MaximumOutput + _MinimumOutput) / 2.0) + _Bias) THEN
			_iTuning := 10;
		ELSIF (NOT bAutoTuning) THEN
			_iTuning := 0;
		END_IF

	10: (* setup *)
		_AutoTuning.fSetY	:= _MaximumOutput;
		_AutoTuning.tTimeout:= tTuningTimeout;
		_AutoTuning.fMinY	:= _MinimumOutput;
		_AutoTuning.fMaxY	:= _MaximumOutput;
		_AutoTuning.fDeadband:= _Deadband;
		_AutoTuning.eMode	:= eTuningMode;
		_iTuning := 20;

	20: (* wait busy *)
		_AutoTuning.bStart := TRUE;
		IF _AutoTuning.bAborted THEN
			_iTuning := 200;
		ELSIF _AutoTuning.bBusy THEN
			_iTuning := 30;
		END_IF

	30: (* wait done *)
		IF _AutoTuning.bAborted THEN
			_iTuning := 200;
		ELSIF _AutoTuning.bDone THEN
			_iTuning := 40;
		END_IF

	40: (* write properties *)
		IF Device.stAdsConn.bValid THEN
			_iTuning := 41;
			_WriteProp(bExecute := FALSE);
			IF (eMode = BACnetLoopMode_Ideal) THEN
				_fTuneKp := _AutoTuning.fPID_Kp;
				_fTuneKi := _AutoTuning.fPID_Ki;
				_fTuneKd := _AutoTuning.fPID_Kd;
			ELSE
				_fTuneKp := _AutoTuning.fPID_Kp;
				IF (_AutoTuning.fPID_Ki <> 0.0) THEN
					_fTuneKi := _fTuneKp / _AutoTuning.fPID_Ki;
				ELSE
					_fTuneKi := 0.0;
				END_IF
				IF (_fTuneKp <> 0.0) THEN
					_fTuneKd := _AutoTuning.fPID_Kd / _fTuneKp;
				ELSE
					_fTuneKd := 0.0;
				END_IF
			END_IF
		ELSE
			_iTuning := 200;
		END_IF

	41: (* write Kp *)
		_WriteProp.DataType	:= BACnetDataType_Real;
		_WriteProp.ptrValue	:= ADR(_fTuneKp);
		_WriteProp.nLenValue:= SIZEOF(_fTuneKp);
		_WriteProp(
			bExecute := TRUE,
			PropertyID := BACnetPropertyIdentifier_ProportionalConstant);
		IF (NOT _WriteProp.bBusy) THEN
			IF (_WriteProp.bError) THEN
				_iTuning := 200;
			ELSE
				_iTuning := 42;
			END_IF
			_WriteProp(bExecute := FALSE);
		END_IF

	42: (* write Ki *)
		_WriteProp.DataType	:= BACnetDataType_Real;
		_WriteProp.ptrValue	:= ADR(_fTuneKi);
		_WriteProp.nLenValue:= SIZEOF(_fTuneKi);
		_WriteProp(
			bExecute := TRUE,
			PropertyID := BACnetPropertyIdentifier_IntegralConstant);
		IF (NOT _WriteProp.bBusy) THEN
			IF (_WriteProp.bError) THEN
				_iTuning := 200;
			ELSE
				_iTuning := 43;
			END_IF
			_WriteProp(bExecute := FALSE);
		END_IF

	43: (* write Kd *)
		_WriteProp.DataType	:= BACnetDataType_Real;
		_WriteProp.ptrValue	:= ADR(_fTuneKd);
		_WriteProp.nLenValue:= SIZEOF(_fTuneKd);
		_WriteProp(
			bExecute := TRUE,
			PropertyID := BACnetPropertyIdentifier_DerivativeConstant);
		IF (NOT _WriteProp.bBusy) THEN
			IF (_WriteProp.bError) THEN
				_iTuning := 200;
			ELSE
				_iTuning := 44;
			END_IF
			_WriteProp(bExecute := FALSE);
		END_IF

	44: (* write Action *)
		_WriteProp.DataType	:= BACnetDataType_Enumerated;
		_WriteProp.ptrValue	:= ADR(_AutoTuning.eAction);
		_WriteProp.nLenValue:= SIZEOF(_AutoTuning.eAction);
		_WriteProp(
			bExecute := TRUE,
			PropertyID := BACnetPropertyIdentifier_Action);
		IF (NOT _WriteProp.bBusy) THEN
			IF (_WriteProp.bError) THEN
				_iTuning := 200;
			ELSE
				_iTuning := 100;
			END_IF
			_WriteProp(bExecute := FALSE);
		END_IF


	100: (* done *)
		IF NOT bAutoTuning THEN
			_iTuning := 0;
		END_IF

	200: (* aborted *)
		IF NOT bAutoTuning THEN
			_iTuning := 0;
		END_IF

END_CASE

(* call auto tuning function block *)
_AutoTuning(
	bStart	:= ,
	bStop	:=	_StatusFlagsBits.out_of_service
			OR	(_Reliability <> BACnetReliability_no_fault_detected),
	fSetY	:= ,
	fDeadband	:= ,
	fX		:= _ControlledVariableValue,
	tTimeout:= ,
	fMinY	:= ,
	fMaxY	:= ,
	fCycleTime := _cycleTime,
	fY		:= _fbAccLimit.X,
	fPID_Kp	=> ,
	fPID_Ki	=> ,
	fPID_Kd	=> ,
	eAction => ,
	bSetY	=> ,
	bWaitY	=> ,
	bWaitX	=> ,
	bReady	=> ,
	bBusy	=> ,
	bDone	=> ,
	bAborted=> bTuningAborted,
	bTimeout=> );

(* set auto tuning state *)
bTuningWaitPV	:= (_iTuning = 5);
bTuningWaitCV	:= (_iTuning > 5 AND _iTuning <= 30);
bTuningAborted	:= (_iTuning = 200);
bTuningActive	:= (_iTuning > 0) AND (NOT bTuningAborted);
bTuningDone		:= (_iTuning = 100);
(* set error info *)
IF (bTuningActive OR bTuningAborted) THEN
	IF (NOT Device.stAdsConn.bValid) THEN
		nErrorId	:= BACnet_ERR_INVALID_ADS_CONN;
	ELSIF _WriteProp.bError THEN
		nErrorId	:= BACnet_ERR_ADS_Write;
	END_IF
END_IF

(* limit present value *)
_fbAccLimit(
	X	:= ,
	Amax:= fAccLimit,
	Tcycle:= _cycleTime,
	Y	=> _PresentValueQ,
	A	=> );

(* calculate proportional band *)
IF (_MaximumOutput > 0.0) AND (_MinimumOutput >= 0.0) THEN
	fPropBand := ((_PresentValueQ - _MinimumOutput) / (_MaximumOutput - _MinimumOutput)) * 100.0;
ELSIF (_MaximumOutput <= 0.0) AND (_MinimumOutput < 0.0) THEN
	fPropBand := ((_PresentValueQ - _MaximumOutput) / (_MaximumOutput - _MinimumOutput)) * 100.0;
ELSIF (_PresentValueQ > 0.0) AND (_MaximumOutput > 0.0) THEN
	fPropBand := (_PresentValueQ / _MaximumOutput) * 100.0;
ELSIF (_PresentValueQ < 0.0) AND (_MinimumOutput < 0.0) THEN
	fPropBand := (_PresentValueQ / _MinimumOutput) * -100.0;
ELSE
	fPropBand := 0.0;
END_IF

(* set error flag *)
bError := (nErrorId <> BACnet_ERR_NO_ERROR);
END_FUNCTION_BLOCK

(* POU FB_BACnet_MultiStateInput, ST *)
FUNCTION_BLOCK FB_BACnet_MultiStateInput
VAR_IN_OUT
	Device	: FB_BACnet_Device;
END_VAR
VAR_OUTPUT
	bReady			: BOOL;
	nPresentValue	: UDINT;
	bOverridden		: BOOL;
	bOutOfService	: BOOL;
	bFault			: BOOL;
	bInAlarm		: BOOL;
	bError			: BOOL;
	nErrorId		: UINT;
END_VAR
VAR
	_PresentValue AT%I*: UDINT; 	(* ~(BACnet_PresentValue 	:		: )
								   		(BACnet_ObjectType 		: MI	: )	*)
	_StatusFlags AT%I*: WORD; 		(* ~(BACnet_StatusFlags 	:		: )	*)
	_StatusFlagsBits : ST_BACnet_StatusFlags;

	_nUpdateCount : UDINT := 0;
END_VAR
(* update server device *)
IF (Device._nUpdateCount = _nUpdateCount) THEN
	Device();
END_IF
(* remind current number of update counter *)
_nUpdateCount := Device._nUpdateCount;

(* check BitString format of StatusFlags --> if StatusFlags are less than 4, object isn't linked correctly *)
IF (_StatusFlags < 4) THEN
	(* wrong mapping *)
	nErrorId := BACnet_ERR_WRONG_MAPPING;
	bReady := FALSE;

ELSIF Device.bOperational THEN
	(* ready state *)
	bReady := TRUE;
	nErrorId := BACnet_ERR_NO_ERROR;

	(* present value *)
	nPresentValue := _PresentValue;

	(* build bit states *)
	_StatusFlagsBits := F_BACnet_StatusFlags(_StatusFlags);

	(* copy states to output *)
	bOverridden := _StatusFlagsBits.overridden;
	bOutOfService := _StatusFlagsBits.out_of_service;
	bFault := _StatusFlagsBits.fault;
	bInAlarm := _StatusFlagsBits.in_alarm;

ELSE
	(* server device not ready, reset local ready also *)
	bReady := FALSE;
	nErrorId := BACnet_ERR_OPERATIONAL;
END_IF
(* set error flag *)
bError := (nErrorId <> BACnet_ERR_NO_ERROR);
END_FUNCTION_BLOCK

(* POU FB_BACnet_MultiStateInput_EX, ST *)
FUNCTION_BLOCK FB_BACnet_MultiStateInput_EX
VAR_IN_OUT
	Device				: FB_BACnet_Device;
END_VAR
VAR_OUTPUT
	bReady				: BOOL;
	nPresentValue		: UDINT;
	bOverridden			: BOOL;
	bOutOfService		: BOOL;
	bFault				: BOOL;
	bInAlarm			: BOOL;
	bOverRange			: BOOL;
	bUnderRange			: BOOL;
	bNoSensor			: BOOL;
	bOpenLoop			: BOOL;
	bShortedLoop		: BOOL;
	bMultiStateFault	: BOOL;
	bOtherFault			: BOOL;
	eEventState			: E_BACNETEVENTSTATE;
	bAckedTrans_ToOffNormal : BOOL;
	bAckedTrans_ToFault		: BOOL;
	bAckedTrans_ToNormal	: BOOL;
	nNbrOfStates		: UDINT;
	tObjectID			: T_BACnet_ObjectIdentifier := 16#FFFFFFFF;
	bError				: BOOL;
	nErrorId			: UINT;
END_VAR
VAR
	_PresentValue AT%I*: UDINT; 		(* ~(BACnet_PresentValue 	:		: )
								   			(BACnet_ObjectType 		: MI	: )	*)
	_NumberOfStates AT%I*: UDINT;		(* ~(BACnet_NumberOfStates	:		: )	*)
	_ObjectId AT%I*: DWORD;				(* ~(BACnet_ObjectIdentifier:		: LINK) *)
	_StatusFlags AT%I*: WORD; 			(* ~(BACnet_StatusFlags 	:		: )	*)
	_EventState AT%I*: WORD; 			(* ~(BACnet_EventState 		:		: )	*)
	_Reliability AT%I*: WORD; 			(* ~(BACnet_Reliability 	:		: )	*)
	_AckedTransitions AT%I*:WORD;		(* ~(BACnet_AckedTransitions:		: ) *)
	_AckedTransBits : ST_BACnet_EventTransitionBits;
	_nUpdateCount : UDINT := 0;
	_StatusFlagsBits : ST_BACnet_StatusFlags;
END_VAR
(* update server device *)
IF (Device._nUpdateCount = _nUpdateCount) THEN
	Device();
END_IF
(* remind current number of update counter *)
_nUpdateCount := Device._nUpdateCount;

(* check object type *)
IF (F_BACnet_GetObjType(_ObjectId) <> BACnetObjectType_MultiStateInput) THEN
	(* wrong mapping / invalid object ID *)
	IF _ObjectId = 0 THEN
		nErrorId := BACnet_ERR_WRONG_MAPPING;
	ELSE
		nErrorId := BACnet_ERR_INVALID_OBJECTID;
	END_IF
	bReady := FALSE;

ELSIF (_StatusFlags < 4) THEN
	(* wrong mapping *)
	nErrorId := BACnet_ERR_WRONG_MAPPING;
	bReady := FALSE;

ELSIF Device.bOperational THEN
	(* ready state *)
	bReady := TRUE;
	nErrorId := BACnet_ERR_NO_ERROR;

	(* present value *)
	nPresentValue := _PresentValue;

	(* build bit states *)
	_StatusFlagsBits := F_BACnet_StatusFlags(_StatusFlags);
	_AckedTransBits		:= F_BACnet_EventTransitionFlags(_AckedTransitions);

	(* copy states to output *)
	bOverridden := _StatusFlagsBits.overridden;
	bOutOfService := _StatusFlagsBits.out_of_service;
	bFault := _StatusFlagsBits.fault;
	bInAlarm := _StatusFlagsBits.in_alarm;
	bOverRange := (_Reliability = BACnetReliability_over_range);
	bUnderRange := (_Reliability = BACnetReliability_under_range);
	bNoSensor := (_Reliability = BACnetReliability_no_sensor);
	bOpenLoop := (_Reliability = BACnetReliability_open_loop);
	bShortedLoop := (_Reliability = BACnetReliability_shorted_loop);
	bMultiStateFault := (_Reliability = BACnetReliability_multi_state_fault);
	bOtherFault := (_Reliability = BACnetReliability_unreliable_other);
	bAckedTrans_ToOffNormal := _AckedTransBits.to_offnormal;
	bAckedTrans_ToFault := _AckedTransBits.to_fault;
	bAckedTrans_ToNormal := _AckedTransBits.to_normal;
	tObjectID := _ObjectId;

	(* convert enumeration *)
	eEventState := _EventState;

	(* number of states *)
	nNbrOfStates := _NumberOfStates;

ELSE
	(* server device not ready, reset local ready also *)
	bReady := FALSE;
	nErrorId := BACnet_ERR_OPERATIONAL;
END_IF
(* set error flag *)
bError := (nErrorId <> BACnet_ERR_NO_ERROR);
END_FUNCTION_BLOCK

(* POU FB_BACnet_MultiStateInput_RAW, ST *)
FUNCTION_BLOCK FB_BACnet_MultiStateInput_RAW
VAR_INPUT
	nRawIn				AT%Q*: DWORD; (* ~(BACnet_PresentValue : : ) *)
	bNoSensor		: BOOL;
	bOverRange		: BOOL;
	bUnderRange		: BOOL;
	bOpenLoop		: BOOL;
	bShortedLoop	: BOOL;
	bCommFailure	: BOOL;
	bOtherFault		: BOOL;
END_VAR
VAR_IN_OUT
	Device				: FB_BACnet_Device;
END_VAR
VAR_OUTPUT
	bReady				: BOOL;
	nPresentValue		: UDINT;
	bOverridden			: BOOL;
	bOutOfService		: BOOL;
	bFault				: BOOL;
	bInAlarm			: BOOL;
	bAckedTrans_ToOffNormal : BOOL;
	bAckedTrans_ToFault		: BOOL;
	bAckedTrans_ToNormal	: BOOL;
	nNbrOfStates		: UDINT;
	bError				: BOOL;
	nErrorId			: UINT;
END_VAR
VAR
	_Reliability AT%Q*: WORD := BACnetReliability_no_fault_detected;(* ~(BACnet_Reliability 	:		: )	*)
	_PresentValue AT%I*: UDINT; 		(* ~(BACnet_PresentValue 	:		: )
								   			(BACnet_ObjectType 		: MI	: )	*)
	_NumberOfStates AT%I*: UDINT;		(* ~(BACnet_NumberOfStates	:		: )	*)
	_ObjectId AT%I*: DWORD;				(* ~(BACnet_ObjectIdentifier:		: LINK) *)
	_StatusFlags AT%I*: WORD; 			(* ~(BACnet_StatusFlags 	:		: )	*)
	_AckedTransitions AT%I*:WORD;		(* ~(BACnet_AckedTransitions:		: ) *)
	_AckedTransBits : ST_BACnet_EventTransitionBits;
	_nUpdateCount : UDINT := 0;
	_StatusFlagsBits : ST_BACnet_StatusFlags;
END_VAR
(* update server device *)
IF (Device._nUpdateCount = _nUpdateCount) THEN
	Device();
END_IF
(* remind current number of update counter *)
_nUpdateCount := Device._nUpdateCount;

(* handle raw error *)
IF bNoSensor THEN
	_Reliability := BACnetReliability_no_sensor;
ELSIF bOverRange THEN
	_Reliability := BACnetReliability_over_range;
ELSIF bUnderRange THEN
	_Reliability := BACnetReliability_under_range;
ELSIF bOpenLoop THEN
	_Reliability := BACnetReliability_open_loop;
ELSIF bShortedLoop THEN
	_Reliability := BACnetReliability_shorted_loop;
ELSIF bCommFailure THEN
	_Reliability := BACnetReliability_communication_failure;
ELSIF bOtherFault THEN
	_Reliability := BACnetReliability_unreliable_other;
ELSE
	_Reliability := BACnetReliability_no_fault_detected;
END_IF

(* check object type *)
IF (F_BACnet_GetObjType(_ObjectId) <> BACnetObjectType_MultiStateInput) THEN
	(* wrong mapping / invalid object ID *)
	IF _ObjectId = 0 THEN
		nErrorId := BACnet_ERR_WRONG_MAPPING;
	ELSE
		nErrorId := BACnet_ERR_INVALID_OBJECTID;
	END_IF
	bReady := FALSE;

ELSIF (_StatusFlags < 4) THEN
	(* wrong mapping *)
	nErrorId := BACnet_ERR_WRONG_MAPPING;
	bReady := FALSE;

ELSIF Device.bOperational THEN
	(* ready state *)
	bReady := TRUE;
	nErrorId := BACnet_ERR_NO_ERROR;

	(* present value *)
	nPresentValue := _PresentValue;

	(* build bit states *)
	_StatusFlagsBits := F_BACnet_StatusFlags(_StatusFlags);
	_AckedTransBits		:= F_BACnet_EventTransitionFlags(_AckedTransitions);

	(* copy states to output *)
	bOverridden := _StatusFlagsBits.overridden;
	bOutOfService := _StatusFlagsBits.out_of_service;
	bFault := _StatusFlagsBits.fault;
	bInAlarm := _StatusFlagsBits.in_alarm;
	bAckedTrans_ToOffNormal := _AckedTransBits.to_offnormal;
	bAckedTrans_ToFault := _AckedTransBits.to_fault;
	bAckedTrans_ToNormal := _AckedTransBits.to_normal;

	(* number of states *)
	nNbrOfStates := _NumberOfStates;

ELSE
	(* server device not ready, reset local ready also *)
	bReady := FALSE;
	nErrorId := BACnet_ERR_OPERATIONAL;
END_IF
(* set error flag *)
bError := (nErrorId <> BACnet_ERR_NO_ERROR);
END_FUNCTION_BLOCK

(* POU FB_BACnet_MultiStateOutput, ST *)
FUNCTION_BLOCK FB_BACnet_MultiStateOutput
VAR_INPUT
	bEnablePV		: BOOL; (* enable present value with priority x in priority array, FALSE = priority x disable *)
	bNullPV			: BOOL; (* clear priority entry *)
	nPV				: UDINT; (* number for priority x, when input bEnablePV is TRUE *)
END_VAR
VAR_IN_OUT
	Device	: FB_BACnet_Device;
END_VAR
VAR_OUTPUT
	bReady			: BOOL;
	nPresentValue	: UDINT;
	bOverridden		: BOOL;
	bOutOfService	: BOOL;
	bFault			: BOOL;
	bInAlarm		: BOOL;
	nNbrOfStates	: UDINT;
	bError			: BOOL;
	nErrorId		: UINT;
END_VAR
VAR
	_PresentValue AT%I*: UDINT; 			(* ~(BACnet_PresentValue 		:		: )
								   				(BACnet_ObjectType			: MO	: )	*)
	_NumberOfStates AT%I*: UDINT;			(* ~(BACnet_NumberOfStates		:		: )	*)
	_StatusFlags AT%I*: WORD; 				(* ~(BACnet_StatusFlags			:		: )	*)
    _PresentValue_Priority12 AT%Q*: UDINT;	(* ~(BACnet_PresentValue_Priority12:	: )	*)
	_StatusFlagsBits : ST_BACnet_StatusFlags;
	_nUpdateCount : UDINT := 0;
END_VAR
(* update server device *)
IF (Device._nUpdateCount = _nUpdateCount) THEN
	Device();
END_IF
(* remind current number of update counter *)
_nUpdateCount := Device._nUpdateCount;

IF Device.bFirstCycle THEN
	(* first call of the server device since reboot/reset *)
	bReady := FALSE;
	_PresentValue_Priority12 := 16#FFFFFFFF;

ELSIF (_StatusFlags < 4) THEN
	(* wrong mapping *)
	nErrorId := BACnet_ERR_WRONG_MAPPING;
	bReady := FALSE;

ELSIF Device.bOperational THEN
	(* ready state *)
	bReady := TRUE;
	nErrorId := BACnet_ERR_NO_ERROR;

	(* write into priority array *)
	_PresentValue_Priority12 := F_BACnet_MultiStatePV(bEnablePV, bNullPV, nPV);

	(* present value *)
	nPresentValue := _PresentValue;

	(* build bit states *)
	_StatusFlagsBits := F_BACnet_StatusFlags(_StatusFlags);

	(* copy states to output *)
	bOverridden := _StatusFlagsBits.overridden;
	bOutOfService := _StatusFlagsBits.out_of_service;
	bFault := _StatusFlagsBits.fault;
	bInAlarm := _StatusFlagsBits.in_alarm;

	(* number of states *)
	nNbrOfStates := _NumberOfStates;

ELSE
	(* server device not ready, reset local ready also *)
	bReady := FALSE;
	nErrorId := BACnet_ERR_OPERATIONAL;
END_IF
(* set error flag *)
bError := (nErrorId <> BACnet_ERR_NO_ERROR);
END_FUNCTION_BLOCK

(* POU FB_BACnet_MultiStateOutput_ADS, ST *)
FUNCTION_BLOCK FB_BACnet_MultiStateOutput_ADS
VAR_INPUT
	bEnablePV			: BOOL; (* enable PV write commands *)
	bNullPV				: BOOL; (* clear priority entry *)
	nPV					: UDINT; (* number for priority x, when input bEnablePV is TRUE and bNullPV is FALSE *)
	bManual				: BOOL; (* FALSE --> TRUE: write present_value immediately, FALSE: only write present_value on-change, TRUE: write present_value on-change and when device turns operational *)
	ePriority			: E_BACNETPRIORITY := BACNETPRIORITY_12;
END_VAR
VAR_IN_OUT
	Device				: FB_BACnet_Device;
END_VAR
VAR_OUTPUT
	bReady				: BOOL;
	bPvDone				: BOOL; (* present_value written over ADS *)
	nPresentValue		: UDINT;
	bOverridden			: BOOL;
	bOutOfService		: BOOL;
	bFault				: BOOL;
	bInAlarm			: BOOL;
	nNbrOfStates		: UDINT;
	tObjectID			: T_BACnet_ObjectIdentifier := 16#FFFFFFFF;
	bError				: BOOL;
	nErrorId			: UINT;
	nAdsErrorId			: UDINT;
END_VAR
VAR
	_StatusFlags AT%I*: WORD; 				(* ~(BACnet_StatusFlags			:		: )	*)
	_PresentValue AT%I*: UDINT; 			(* ~(BACnet_PresentValue 		:		: )
								   				(BACnet_ObjectType			: MO	: )	*)
	_NumberOfStates AT%I*: UDINT;			(* ~(BACnet_NumberOfStates		:		: )	*)
	_ObjectId AT%I*: DWORD;					(* ~(BACnet_ObjectIdentifier	:		: LINK) *)
	_StatusFlagsBits : ST_BACnet_StatusFlags;
    _PresentValue_Ads : UDINT;
	_nUpdateCount : UDINT := 0;
	_WriteProp : FB_BACnet_WriteProp;
	_rtrigManual : R_TRIG;
	_bNullPvOld : BOOL;
	_nObjType : E_BACNETOBJECTTYPE;
END_VAR
(* update server device *)
IF (Device._nUpdateCount = _nUpdateCount) THEN
	Device();
END_IF
(* remind current number of update counter *)
_nUpdateCount := Device._nUpdateCount;

(* trigger on manual flag *)
_rtrigManual(CLK:= bManual, Q=> );

(* decode object type *)
_nObjType := F_BACnet_GetObjType(_ObjectId);

IF Device.bFirstCycle THEN
	(* first call of the server device since reboot/reset *)
	bReady := FALSE;
	bPvDone := FALSE;

ELSIF _nObjType <> BACnetObjectType_MultiStateOutput THEN
	(* wrong mapped object type *)
	nErrorId := BACnet_ERR_INVALID_OBJECTTYPE;
	bReady := FALSE;
	bPvDone := FALSE;

ELSIF (_StatusFlags < 4) THEN
	(* wrong mapping *)
	nErrorId := BACnet_ERR_WRONG_MAPPING;
	bReady := FALSE;
	bPvDone := FALSE;

ELSIF Device.bOperational THEN

	IF Device.stAdsConn.bValid THEN
		(* write present_value on manual trigger, on-change and on operational recover *)
		IF		bEnablePV
			AND	(		_rtrigManual.Q
					OR	(nPV <> _PresentValue_Ads)
					OR	((NOT bReady) AND bManual)
					OR	(bNullPV <> _bNullPvOld)
				)
		THEN
			_WriteProp.bExecute := TRUE;
			bPvDone := FALSE;
			(* write depending on enable state *)
			IF bNullPV THEN
				_PresentValue_Ads := 0;
			ELSE
				_PresentValue_Ads := nPV;
			END_IF
			_bNullPvOld := bNullPV;
		END_IF

		(* ready state *)
		IF (nAdsErrorId = 0) THEN
			bReady := TRUE;
			nErrorId := BACnet_ERR_NO_ERROR;
		END_IF

	ELSE
		(* invalid ADS connection *)
		bReady := FALSE;
		nErrorId := BACnet_ERR_INVALID_ADS_CONN;
		bPvDone := FALSE;
	END_IF

	(* present value *)
	nPresentValue := _PresentValue;

	(* build bit states *)
	_StatusFlagsBits := F_BACnet_StatusFlags(_StatusFlags);

	(* copy states to output *)
	bOverridden := _StatusFlagsBits.overridden;
	bOutOfService := _StatusFlagsBits.out_of_service;
	bFault := _StatusFlagsBits.fault;
	bInAlarm := _StatusFlagsBits.in_alarm;
	tObjectID := _ObjectId;

	(* number of states *)
	nNbrOfStates := _NumberOfStates;

ELSE
	(* server device not ready, reset local ready also *)
	bReady := FALSE;
	nErrorId := BACnet_ERR_OPERATIONAL;
	bPvDone := FALSE;
END_IF

(* call write property command *)
_WriteProp(
	BACnetDevicePort	:= Device.stAdsConn.nAmsPort,
	bExecute			:= ,
	sNetId				:= Device.stAdsConn.sAmsNetId,
	ObjectType			:= _nObjType,
	PropertyID			:= BACnetPropertyIdentifier_PresentValue,
	Priority			:= ePriority,
	DataType			:= BACnetDataType_UnsignedInteger,
	ObjectInstance		:= F_BACnet_GetObjInstance(_ObjectId),
	ptrValue			:= ADR(_PresentValue_Ads),
	nLenValue			:= SIZEOF(_PresentValue_Ads),
	bDone				=> ,
	bBusy				=> ,
	bError				=> ,
	nErrID				=> );

(* set done flag *)
IF _WriteProp.bExecute AND (NOT _WriteProp.bBusy) THEN
	(* check if command was finished with error *)
	IF _WriteProp.bError THEN
		bPvDone		:= FALSE;
		bReady		:= FALSE;
		nErrorId	:= BACnet_ERR_ADS_Write;
	ELSE
		(* successful written *)
		bPvDone		:= TRUE;
	END_IF
	nAdsErrorId := _WriteProp.nErrID;
	(* reset execution bit *)
	_WriteProp(bExecute := FALSE);
END_IF

(* set error flag *)
bError := (nErrorId <> BACnet_ERR_NO_ERROR) OR (nAdsErrorId <> 0);
END_FUNCTION_BLOCK

